KUKA KRL program: MyProgram_048().src

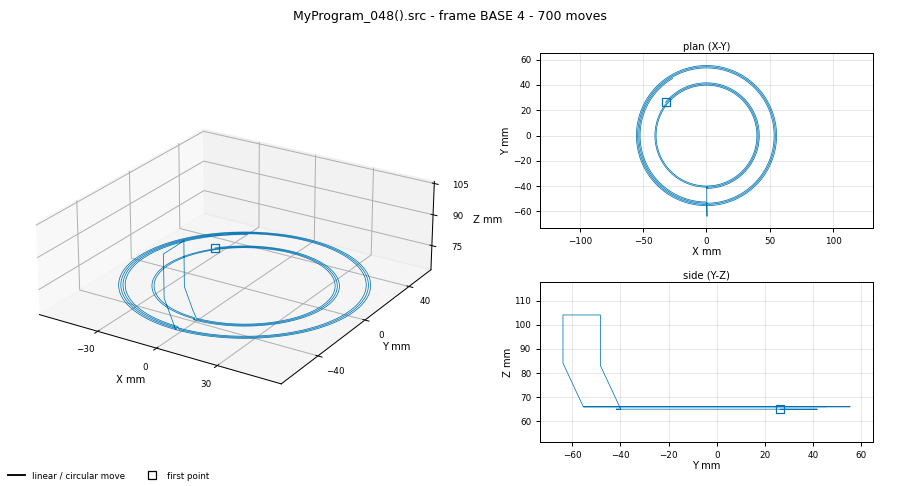
[picture p0: tool path of MyProgram_048().src in frame BASE 4, 700 of 700 moves have a stored position in this frame; points joined in program order, loops and branches not executed]
&ACCESS RVP
&REL 1
&PARAM TEMPLATE = C:\KRC\Roboter\Template\vorgabe
&PARAM EDITMASK = *
DEF MyProgram_048()
; ---- Setting reference (Base) ----
$BASE = BASE_DATA[4]

; --------------------------
; ---- Setting tool (TCP) ----
$TOOL = TOOL_DATA[3]
; --------------------------

$VEL.CP = VEL_APROX_PRINT
Startdeposition()
$VEL.CP = VEL_PRINT
LIN {X -32.3205,Y 26.3963,Z 65,A 132.8032,B 24.8389,C -2.9281,E1 24.8778,E2 -49.5424} C_DIS
LIN {X -30.8175,Y 28.1363,Z 65,A 129.9758,B 24.8376,C -2.9396,E1 24.8831,E2 -46.7299} C_DIS
LIN {X -29.3729,Y 29.641,Z 65,A 126.9235,B 24.8371,C -2.9443,E1 24.889,E2 -43.6757} C_DIS
LIN {X -27.5809,Y 31.3158,Z 65,A 123.4844,B 24.8363,C -2.951,E1 24.8961,E2 -40.2389} C_DIS
LIN {X -25.6579,Y 32.9102,Z 65,A 120.0277,B 24.8356,C -2.9579,E1 24.9037,E2 -36.7858} C_DIS
LIN {X -22.8662,Y 34.9072,Z 65,A 115.1658,B 24.8347,C -2.9653,E1 24.9148,E2 -31.9251} C_DIS
LIN {X -20.5395,Y 36.3254,Z 65,A 111.0714,B 24.8345,C -2.9676,E1 24.9247,E2 -27.824} C_DIS
LIN {X -17.2944,Y 37.9774,Z 65,A 106.8541,B 24.8325,C -2.9849,E1 24.9352,E2 -23.6369} C_DIS
LIN {X -15.0192,Y 38.9331,Z 65,A 102.7286,B 24.8331,C -2.9804,E1 24.946,E2 -19.4915} C_DIS
LIN {X -12.6961,Y 39.7516,Z 65,A 99.3773,B 24.8326,C -2.9847,E1 24.9548,E2 -16.1444} C_DIS
LIN {X -10.2597,Y 40.4489,Z 65,A 96.7038,B 24.831,C -2.9984,E1 24.962,E2 -13.4995} C_DIS
LIN {X -8.3518,Y 40.8853,Z 65,A 93.3297,B 24.8318,C -2.9918,E1 24.9712,E2 -10.1056} C_DIS
LIN {X -5.0291,Y 41.4254,Z 65,A 88.9173,B 24.8311,C -2.9975,E1 24.9834,E2 -5.7032} C_DIS
LIN {X -2.4514,Y 41.657,Z 65,A 85.2136,B 24.8311,C -2.9971,E1 24.9937,E2 -1.9969} C_DIS
LIN {X -0.4444,Y 41.7276,Z 65,A 82.0555,B 24.8317,C -2.9923,E1 25.0026,E2 1.1727} C_DIS
LIN {X 3.7427,Y 41.5615,Z 65,A 77.3936,B 24.83,C -3.0075,E1 25.0155,E2 5.7968} C_DIS
LIN {X 5.9938,Y 41.297,Z 65,A 73.4068,B 24.8315,C -2.9945,E1 25.0266,E2 9.8111} C_DIS
LIN {X 8.6502,Y 40.8239,Z 65,A 69.8403,B 24.8315,C -2.9949,E1 25.0363,E2 13.3725} C_DIS
LIN {X 11.6644,Y 40.0663,Z 65,A 65.7716,B 24.8314,C -2.9951,E1 25.0473,E2 17.4342} C_DIS
LIN {X 14.4066,Y 39.164,Z 65,A 62.3461,B 24.8309,C -2.9997,E1 25.0563,E2 20.8419} C_DIS
LIN {X 15.9978,Y 38.5419,Z 65,A 59.5196,B 24.8319,C -2.9903,E1 25.0636,E2 23.6845} C_DIS
LIN {X 19.3949,Y 36.9485,Z 65,A 55.141,B 24.8313,C -2.9959,E1 25.0746,E2 28.0383} C_DIS
LIN {X 21.1243,Y 35.988,Z 65,A 51.5538,B 24.8332,C -2.9788,E1 25.0834,E2 31.6554} C_DIS
LIN {X 23.0276,Y 34.8007,Z 65,A 48.6817,B 24.8334,C -2.9773,E1 25.0901,E2 34.5218} C_DIS
LIN {X 24.9284,Y 33.4655,Z 65,A 45.4862,B 24.834,C -2.9719,E1 25.0974,E2 37.7189} C_DIS
LIN {X 26.8036,Y 31.9836,Z 65,A 42.1697,B 24.8347,C -2.9653,E1 25.1046,E2 41.0384} C_DIS
LIN {X 28.6861,Y 30.3064,Z 65,A 38.7348,B 24.8355,C -2.9589,E1 25.1116,E2 44.4745} C_DIS
LIN {X 30.3503,Y 28.6394,Z 65,A 35.6045,B 24.836,C -2.9538,E1 25.1177,E2 47.6035} C_DIS
LIN {X 31.8657,Y 26.9436,Z 65,A 32.0272,B 24.8376,C -2.9395,E1 25.1243,E2 51.1986} C_DIS
LIN {X 33.4817,Y 24.9072,Z 65,A 28.9748,B 24.8376,C -2.9395,E1 25.1294,E2 54.2366} C_DIS
LIN {X 34.85,Y 22.9529,Z 65,A 25.5823,B 24.8387,C -2.9294,E1 25.1348,E2 57.6362} C_DIS
LIN {X 35.9583,Y 21.1746,Z 65,A 22.8285,B 24.8393,C -2.924,E1 25.1388,E2 60.3887} C_DIS
LIN {X 36.8509,Y 19.5803,Z 65,A 20.2123,B 24.8403,C -2.9156,E1 25.1423,E2 63.0112} C_DIS
LIN {X 38.143,Y 16.9264,Z 65,A 16.3814,B 24.8411,C -2.9081,E1 25.1468,E2 66.839} C_DIS
LIN {X 38.9023,Y 15.0995,Z 65,A 13.8688,B 24.8416,C -2.9039,E1 25.1494,E2 69.3479} C_DIS
LIN {X 39.6903,Y 12.8856,Z 65,A 10.013,B 24.8437,C -2.8839,E1 25.1529,E2 73.2292} C_DIS
LIN {X 40.4156,Y 10.3892,Z 65,A 7.2043,B 24.8435,C -2.8862,E1 25.155,E2 76.0163} C_DIS
LIN {X 40.9346,Y 8.1069,Z 65,A 3.7683,B 24.845,C -2.8727,E1 25.1571,E2 79.4643} C_DIS
LIN {X 41.2614,Y 6.2336,Z 65,A 1.2108,B 24.8457,C -2.8656,E1 25.1582,E2 82.0235} C_DIS
LIN {X 41.531,Y 4.0697,Z 65,A -2.1598,B 24.8474,C -2.8499,E1 25.1593,E2 85.4114} C_DIS
LIN {X 41.6995,Y 1.5955,Z 65,A -5.1201,B 24.8477,C -2.8469,E1 25.1597,E2 88.3612} C_DIS
LIN {X 41.7291,Y 0.1295,Z 65,A -7.4448,B 24.849,C -2.8352,E1 25.1597,E2 90.6997} C_DIS
LIN {X 41.6403,Y -2.7296,Z 65,A -11.1427,B 24.8499,C -2.8268,E1 25.1593,E2 94.3955} C_DIS
LIN {X 41.4605,Y -4.7326,Z 65,A -13.8628,B 24.8507,C -2.8188,E1 25.1585,E2 97.1184} C_DIS
LIN {X 41.1292,Y -7.0549,Z 65,A -17.206,B 24.852,C -2.8066,E1 25.1571,E2 100.4708} C_DIS
LIN {X 40.6295,Y -9.5191,Z 65,A -20.7553,B 24.8533,C -2.7942,E1 25.155,E2 104.0287} C_DIS
LIN {X 39.9708,Y -11.9877,Z 65,A -24.0951,B 24.8542,C -2.7863,E1 25.1524,E2 107.3682} C_DIS
LIN {X 39.1708,Y -14.3878,Z 65,A -27.523,B 24.8552,C -2.7766,E1 25.1493,E2 110.7999} C_DIS
LIN {X 38.33,Y -16.4987,Z 65,A -30.7347,B 24.8563,C -2.7657,E1 25.1458,E2 114.0196} C_DIS
LIN {X 37.2921,Y -18.727,Z 65,A -34.2725,B 24.8576,C -2.7531,E1 25.1415,E2 117.5684} C_DIS
LIN {X 35.9701,Y -21.1546,Z 65,A -37.5233,B 24.8578,C -2.7515,E1 25.1371,E2 120.806} C_DIS
LIN {X 35.1122,Y -22.5497,Z 65,A -40.3199,B 24.8594,C -2.736,E1 25.1329,E2 123.625} C_DIS
LIN {X 33.0565,Y -25.4681,Z 65,A -44.5679,B 24.8596,C -2.7339,E1 25.1259,E2 127.8576} C_DIS
LIN {X 30.9077,Y -28.0379,Z 65,A -50.2918,B 24.8627,C -2.7037,E1 25.1154,E2 133.6271} C_DIS
LIN {X 27.7752,Y -31.1432,Z 65,A -56.1001,B 24.8637,C -2.6938,E1 25.1036,E2 139.4351} C_DIS
LIN {X 25.3244,Y -33.1672,Z 65,A -60.489,B 24.8647,C -2.6842,E1 25.0939,E2 143.8306} C_DIS
LIN {X 22.261,Y -35.2964,Z 65,A -64.6735,B 24.8642,C -2.6892,E1 25.0842,E2 147.9891} C_DIS
LIN {X 20.7403,Y -36.2105,Z 65,A -67.3879,B 24.8651,C -2.6804,E1 25.0777,E2 150.7159} C_DIS
LIN {X 18.6693,Y -37.3207,Z 65,A -70.5143,B 24.8655,C -2.6767,E1 25.0699,E2 153.8425} C_DIS
LIN {X 16.6026,Y -38.2847,Z 65,A -73.9067,B 24.8663,C -2.668,E1 25.0613,E2 157.2473} C_DIS
LIN {X 14.2014,Y -39.2388,Z 65,A -77.1234,B 24.8663,C -2.6683,E1 25.0529,E2 160.4561} C_DIS
LIN {X 12.1209,Y -39.9312,Z 65,A -80.2732,B 24.8669,C -2.6627,E1 25.0445,E2 163.6136} C_DIS
LIN {X 9.9555,Y -40.5247,Z 65,A -83.3276,B 24.8671,C -2.66,E1 25.0362,E2 166.6696} C_DIS
LIN {X 7.6108,Y -41.0292,Z 65,A -86.1957,B 24.8668,C -2.6636,E1 25.0284,E2 169.5257} C_DIS
LIN {X 6.2927,Y -41.2524,Z 65,A -88.5034,B 24.8676,C -2.6553,E1 25.022,E2 171.8509} C_DIS
LIN {X 4.1311,Y -41.525,Z 65,A -91.2129,B 24.8674,C -2.6577,E1 25.0145,E2 174.5529} C_DIS
LIN {X 2.1588,Y -41.6739,Z 65,A -94.0601,B 24.8677,C -2.6546,E1 25.0065,E2 177.4061} C_DIS
LIN {X 0.2084,Y -41.7255,Z 65,A -95.7171,B 24.8663,C -2.6686,E1 25.002,E2 179.0294} C_DIS
Enddeposition()
LIN {X 0.2084,Y -41.7255,Z 65,A -95.7171,B 24.8663,C -2.6686,E1 25.002,E2 179.0294} C_DIS
Startdeposition()
$VEL.CP = VEL_PRINT
LIN {X 0.7849,Y -40.7795,Z 65,A -94.3839,B 24.8639,C -2.6925,E1 25.0059,E2 177.6397} C_DIS
LIN {X 3.4989,Y -40.6375,Z 65,A -90.8703,B 24.8641,C -2.6897,E1 25.0157,E2 174.1342} C_DIS
LIN {X 5.4478,Y -40.4216,Z 65,A -88.0105,B 24.8638,C -2.6929,E1 25.0236,E2 171.2689} C_DIS
LIN {X 7.6059,Y -40.0718,Z 65,A -84.7696,B 24.8633,C -2.6978,E1 25.0325,E2 168.0199} C_DIS
LIN {X 10.1651,Y -39.5001,Z 65,A -81.273,B 24.8633,C -2.6985,E1 25.042,E2 164.5267} C_DIS
LIN {X 12.8249,Y -38.7189,Z 65,A -76.8382,B 24.8619,C -2.7113,E1 25.0539,E2 160.0697} C_DIS
LIN {X 15.5731,Y -37.6976,Z 65,A -73.1485,B 24.8621,C -2.7102,E1 25.0635,E2 156.3906} C_DIS
LIN {X 17.805,Y -36.6959,Z 65,A -69.8338,B 24.8617,C -2.7136,E1 25.0718,E2 153.0764} C_DIS
LIN {X 19.7266,Y -35.6999,Z 65,A -66.6692,B 24.861,C -2.7206,E1 25.0797,E2 149.9041} C_DIS
LIN {X 21.6021,Y -34.5967,Z 65,A -63.8109,B 24.8607,C -2.7231,E1 25.0865,E2 147.049} C_DIS
LIN {X 23.9097,Y -33.0449,Z 65,A -59.7045,B 24.8596,C -2.734,E1 25.0959,E2 142.9308} C_DIS
LIN {X 25.861,Y -31.5412,Z 65,A -56.2483,B 24.8589,C -2.7413,E1 25.1035,E2 139.4702} C_DIS
LIN {X 27.7138,Y -29.926,Z 65,A -53.35,B 24.8589,C -2.74,E1 25.1095,E2 136.5865} C_DIS
LIN {X 28.9865,Y -28.6944,Z 65,A -50.4742,B 24.8577,C -2.7523,E1 25.1152,E2 133.6937} C_DIS
LIN {X 30.4702,Y -27.1136,Z 65,A -47.0406,B 24.8563,C -2.7663,E1 25.1217,E2 130.2422} C_DIS
LIN {X 32.3443,Y -24.8482,Z 65,A -43.3381,B 24.8559,C -2.7698,E1 25.1281,E2 126.5486} C_DIS
LIN {X 33.6292,Y -23.0807,Z 65,A -40.4032,B 24.8553,C -2.7758,E1 25.1329,E2 123.6139} C_DIS
LIN {X 34.9472,Y -21.0305,Z 65,A -36.6735,B 24.8537,C -2.7905,E1 25.1384,E2 119.8682} C_DIS
LIN {X 35.9255,Y -19.3122,Z 65,A -34.0007,B 24.8531,C -2.7966,E1 25.142,E2 117.1948} C_DIS
LIN {X 37.0399,Y -17.0779,Z 65,A -30.6076,B 24.8522,C -2.805,E1 25.1461,E2 113.8003} C_DIS
LIN {X 37.907,Y -15.0554,Z 65,A -27.4857,B 24.8512,C -2.8147,E1 25.1494,E2 110.6725} C_DIS
LIN {X 38.6802,Y -12.9398,Z 65,A -24.7937,B 24.851,C -2.8162,E1 25.1519,E2 107.992} C_DIS
LIN {X 39.2211,Y -11.1934,Z 65,A -22.2257,B 24.8502,C -2.8241,E1 25.154,E2 105.42} C_DIS
LIN {X 39.6949,Y -9.3771,Z 65,A -19.2563,B 24.8487,C -2.838,E1 25.156,E2 102.435} C_DIS
LIN {X 40.1515,Y -7.1725,Z 65,A -16.0267,B 24.8475,C -2.849,E1 25.1577,E2 99.1981} C_DIS
LIN {X 40.5125,Y -4.7251,Z 65,A -12.5987,B 24.8464,C -2.8591,E1 25.159,E2 95.7665} C_DIS
LIN {X 40.7053,Y -2.5869,Z 65,A -9.1965,B 24.8447,C -2.8752,E1 25.1596,E2 92.3463} C_DIS
LIN {X 40.776,Y 0.949,Z 65,A -4.9181,B 24.8443,C -2.8789,E1 25.1596,E2 88.0845} C_DIS
LIN {X 40.615,Y 3.7424,Z 65,A -0.3025,B 24.8417,C -2.9029,E1 25.1587,E2 83.4396} C_DIS
LIN {X 40.2879,Y 6.363,Z 65,A 3.1785,B 24.8408,C -2.9104,E1 25.1573,E2 79.9614} C_DIS
LIN {X 39.6611,Y 9.5174,Z 65,A 7.3091,B 24.8401,C -2.9174,E1 25.1549,E2 75.8382} C_DIS
LIN {X 39.038,Y 11.8165,Z 65,A 10.7303,B 24.8388,C -2.9286,E1 25.1523,E2 72.4102} C_DIS
LIN {X 38.4737,Y 13.5412,Z 65,A 12.883,B 24.8388,C -2.9293,E1 25.1503,E2 70.2679} C_DIS
LIN {X 37.9097,Y 15.0486,Z 65,A 15.4724,B 24.8374,C -2.9413,E1 25.1477,E2 67.6645} C_DIS
LIN {X 36.8271,Y 17.532,Z 65,A 19.3626,B 24.8361,C -2.9532,E1 25.1432,E2 63.7671} C_DIS
LIN {X 35.7144,Y 19.7005,Z 65,A 22.6885,B 24.8353,C -2.9607,E1 25.1388,E2 60.441} C_DIS
LIN {X 34.6226,Y 21.5607,Z 65,A 25.3115,B 24.8351,C -2.9618,E1 25.1351,E2 57.8287} C_DIS
LIN {X 33.0626,Y 23.8852,Z 65,A 29.4017,B 24.8338,C -2.9741,E1 25.1286,E2 53.7296} C_DIS
LIN {X 32.106,Y 25.1559,Z 65,A 32.0073,B 24.8325,C -2.9854,E1 25.1241,E2 51.1095} C_DIS
LIN {X 30.2152,Y 27.3986,Z 65,A 36.0076,B 24.8317,C -2.9927,E1 25.1168,E2 47.1101} C_DIS
LIN {X 28.5261,Y 29.1528,Z 65,A 39.37,B 24.831,C -2.9989,E1 25.1102,E2 43.7473} C_DIS
LIN {X 26.7641,Y 30.7779,Z 65,A 42.6418,B 24.8304,C -3.0039,E1 25.1034,E2 40.4767} C_DIS
LIN {X 24.9657,Y 32.2538,Z 65,A 45.9762,B 24.8296,C -3.0108,E1 25.0961,E2 37.1383} C_DIS
LIN {X 22.9381,Y 33.7259,Z 65,A 49.302,B 24.8293,C -3.0136,E1 25.0885,E2 33.8175} C_DIS
LIN {X 21.1922,Y 34.8494,Z 65,A 52.6119,B 24.8281,C -3.024,E1 25.0806,E2 30.4934} C_DIS
LIN {X 18.538,Y 36.3308,Z 65,A 56.2779,B 24.8285,C -3.0204,E1 25.0717,E2 26.8464} C_DIS
LIN {X 16.757,Y 37.1859,Z 65,A 59.369,B 24.8276,C -3.0283,E1 25.0638,E2 23.7444} C_DIS
LIN {X 14.6433,Y 38.0684,Z 65,A 62.6886,B 24.8271,C -3.033,E1 25.0552,E2 20.4212} C_DIS
LIN {X 12.286,Y 38.8933,Z 65,A 65.5956,B 24.8278,C -3.027,E1 25.0475,E2 17.5339} C_DIS
LIN {X 10.6833,Y 39.3631,Z 65,A 69.197,B 24.8255,C -3.0468,E1 25.0377,E2 13.8914} C_DIS
LIN {X 7.2645,Y 40.135,Z 65,A 73.3488,B 24.8265,C -3.0378,E1 25.0265,E2 9.7661} C_DIS
LIN {X 4.9873,Y 40.4811,Z 65,A 76.4292,B 24.8267,C -3.0364,E1 25.0179,E2 6.6917} C_DIS
LIN {X 3.2904,Y 40.6541,Z 65,A 78.7021,B 24.8269,C -3.0349,E1 25.0116,E2 4.4237} C_DIS
LIN {X 1.2643,Y 40.7675,Z 65,A 82.277,B 24.8257,C -3.0447,E1 25.0016,E2 0.8265} C_DIS
LIN {X -1.7811,Y 40.7482,Z 65,A 86.121,B 24.8266,C -3.0376,E1 24.9909,E2 -3.0011} C_DIS
LIN {X -4.2792,Y 40.562,Z 65,A 90.6441,B 24.8252,C -3.0494,E1 24.9783,E2 -7.5547} C_DIS
LIN {X -8.1041,Y 39.974,Z 65,A 95.7175,B 24.8262,C -3.0404,E1 24.9644,E2 -12.6121} C_DIS
LIN {X -11.7877,Y 39.0471,Z 65,A 100.4469,B 24.8277,C -3.0272,E1 24.9517,E2 -17.3172} C_DIS
LIN {X -14.0402,Y 38.2944,Z 65,A 103.7453,B 24.8283,C -3.0227,E1 24.943,E2 -20.6112} C_DIS
LIN {X -15.9024,Y 37.5593,Z 65,A 106.1998,B 24.8292,C -3.0144,E1 24.9367,E2 -23.0515} C_DIS
LIN {X -18.3667,Y 36.4184,Z 65,A 111.1925,B 24.8282,C -3.023,E1 24.9241,E2 -28.0776} C_DIS
LIN {X -21.3412,Y 34.7588,Z 65,A 115.2173,B 24.8302,C -3.0054,E1 24.9145,E2 -32.0725} C_DIS
LIN {X -23.457,Y 33.3676,Z 65,A 118.8869,B 24.8309,C -2.9999,E1 24.906,E2 -35.7413} C_DIS
LIN {X -25.4735,Y 31.855,Z 65,A 122.4407,B 24.8317,C -2.9927,E1 24.8982,E2 -39.2909} C_DIS
LIN {X -27.3021,Y 30.3017,Z 65,A 125.7452,B 24.8326,C -2.9845,E1 24.8912,E2 -42.5888} C_DIS
LIN {X -29.076,Y 28.6039,Z 65,A 128.9546,B 24.8338,C -2.9737,E1 24.8849,E2 -45.7859} C_DIS
LIN {X -30.3502,Y 27.248,Z 65,A 131.9306,B 24.8341,C -2.9715,E1 24.8792,E2 -48.7696} C_DIS
LIN {X -31.9657,Y 25.3334,Z 65,A 135.4098,B 24.8351,C -2.962,E1 24.8731,E2 -52.2424} C_DIS
LIN {X -33.3945,Y 23.4184,Z 65,A 138.8033,B 24.8361,C -2.9535,E1 24.8676,E2 -55.6321} C_DIS
LIN {X -34.7081,Y 21.4239,Z 65,A 142.1037,B 24.8372,C -2.9437,E1 24.8626,E2 -58.9257} C_DIS
LIN {X -35.7924,Y 19.5577,Z 65,A 145.1702,B 24.8381,C -2.9355,E1 24.8584,E2 -61.9887} C_DIS
LIN {X -36.8745,Y 17.4332,Z 65,A 148.3179,B 24.8394,C -2.9236,E1 24.8545,E2 -65.1249} C_DIS
LIN {X -37.9062,Y 15.0576,Z 65,A 152.2189,B 24.8403,C -2.9157,E1 24.8503,E2 -69.0285} C_DIS
LIN {X -38.711,Y 12.8484,Z 65,A 155.4631,B 24.8414,C -2.9051,E1 24.8473,E2 -72.2657} C_DIS
LIN {X -39.3303,Y 10.8047,Z 65,A 158.6925,B 24.8422,C -2.8984,E1 24.8448,E2 -75.4977} C_DIS
LIN {X -39.881,Y 8.5504,Z 65,A 161.5006,B 24.8438,C -2.8834,E1 24.8431,E2 -78.2865} C_DIS
LIN {X -40.1774,Y 7.0287,Z 65,A 164.2148,B 24.8438,C -2.8824,E1 24.8417,E2 -81.0143} C_DIS
LIN {X -40.5153,Y 4.7009,Z 65,A 167.0069,B 24.8456,C -2.8666,E1 24.8407,E2 -83.7852} C_DIS
LIN {X -40.7269,Y 2.2152,Z 65,A 170.9567,B 24.8463,C -2.8603,E1 24.8399,E2 -87.7438} C_DIS
LIN {X -40.7865,Y -0.2829,Z 65,A 174.5588,B 24.8474,C -2.8503,E1 24.8399,E2 -91.3436} C_DIS
LIN {X -40.6844,Y -2.8956,Z 65,A 178.0933,B 24.8488,C -2.8374,E1 24.8404,E2 -94.8684} C_DIS
LIN {X -40.5292,Y -4.5821,Z 65,A -179.3218,B 24.8493,C -2.8322,E1 24.8411,E2 -97.4565} C_DIS
LIN {X -40.0876,Y -7.5239,Z 65,A -175.1297,B 24.8507,C -2.8196,E1 24.8431,E2 -101.6433} C_DIS
LIN {X -39.5764,Y -9.8657,Z 65,A -171.9067,B 24.8519,C -2.8079,E1 24.8451,E2 -104.8573} C_DIS
LIN {X -38.9417,Y -12.1297,Z 65,A -168.9289,B 24.8533,C -2.7946,E1 24.8474,E2 -107.8205} C_DIS
LIN {X -38.2219,Y -14.2365,Z 65,A -165.2743,B 24.8536,C -2.7914,E1 24.8508,E2 -111.4882} C_DIS
LIN {X -37.2883,Y -16.5297,Z 65,A -161.827,B 24.8547,C -2.7813,E1 24.8546,E2 -114.9305} C_DIS
LIN {X -36.2762,Y -18.6448,Z 65,A -158.6127,B 24.8557,C -2.7715,E1 24.8586,E2 -118.1386} C_DIS
LIN {X -34.9175,Y -21.0801,Z 65,A -154.5325,B 24.8566,C -2.7632,E1 24.8643,E2 -122.22} C_DIS
LIN {X -33.6067,Y -23.1131,Z 65,A -151.0904,B 24.8574,C -2.7552,E1 24.8696,E2 -125.6603} C_DIS
LIN {X -32.3412,Y -24.8523,Z 65,A -147.9387,B 24.858,C -2.7496,E1 24.8749,E2 -128.8136} C_DIS
LIN {X -30.5769,Y -26.9934,Z 65,A -144.1509,B 24.859,C -2.7395,E1 24.8818,E2 -132.5947} C_DIS
LIN {X -28.8359,Y -28.8467,Z 65,A -140.555,B 24.8598,C -2.7323,E1 24.8888,E2 -136.1889} C_DIS
LIN {X -27.004,Y -30.5683,Z 65,A -137.4763,B 24.8611,C -2.72,E1 24.8951,E2 -139.2506} C_DIS
LIN {X -25.0502,Y -32.1887,Z 65,A -133.4236,B 24.8611,C -2.7195,E1 24.9039,E2 -143.3172} C_DIS
LIN {X -23.4292,Y -33.387,Z 65,A -130.3144,B 24.8612,C -2.7183,E1 24.911,E2 -146.4345} C_DIS
LIN {X -20.8855,Y -35.0342,Z 65,A -126.1779,B 24.862,C -2.7106,E1 24.9208,E2 -150.5654} C_DIS
LIN {X -18.5001,Y -36.3502,Z 65,A -122.6394,B 24.8629,C -2.702,E1 24.9295,E2 -154.0934} C_DIS
LIN {X -16.6041,Y -37.2548,Z 65,A -119.5679,B 24.8631,C -2.7003,E1 24.9373,E2 -157.1684} C_DIS
LIN {X -14.3986,Y -38.1611,Z 65,A -116.44,B 24.8637,C -2.6943,E1 24.9454,E2 -160.2887} C_DIS
LIN {X -11.2696,Y -39.1996,Z 65,A -111.5093,B 24.8637,C -2.6948,E1 24.9585,E2 -165.2295} C_DIS
LIN {X -8.4128,Y -39.9106,Z 65,A -107.1405,B 24.8635,C -2.696,E1 24.9704,E2 -169.6068} C_DIS
LIN {X -4.7607,Y -40.5083,Z 65,A -101.7408,B 24.8633,C -2.6977,E1 24.9854,E2 -175.0148} C_DIS
LIN {X -2.1707,Y -40.7293,Z 65,A -98.2739,B 24.8636,C -2.6952,E1 24.995,E2 -178.477} C_DIS
LIN {X 0.2059,Y -40.781,Z 65,A -96.1977,B 24.8653,C -2.678,E1 25.0007,E2 -180.5123} C_DIS
Enddeposition()
LIN {X 0.2059,Y -40.781,Z 65,A -96.1977,B 24.8653,C -2.678,E1 25.0007,E2 -180.5123} C_DIS
Startdeposition()
$VEL.CP = VEL_PRINT
LIN {X -0.4047,Y -39.8429,Z 65,A -97.6468,B 24.8645,C -2.6863,E1 24.9967,E2 -179.0829} C_DIS
LIN {X -2.4418,Y -39.7704,Z 65,A -100.789,B 24.8648,C -2.6832,E1 24.988,E2 -175.9327} C_DIS
LIN {X -4.8574,Y -39.548,Z 65,A -104.0622,B 24.8645,C -2.6864,E1 24.9789,E2 -172.6651} C_DIS
LIN {X -6.9556,Y -39.2329,Z 65,A -107.3,B 24.8646,C -2.6849,E1 24.9699,E2 -169.4206} C_DIS
LIN {X -9.2215,Y -38.7635,Z 65,A -110.5774,B 24.8644,C -2.687,E1 24.961,E2 -166.1442} C_DIS
LIN {X -11.4617,Y -38.1607,Z 65,A -113.8715,B 24.8641,C -2.6897,E1 24.9522,E2 -162.8512} C_DIS
LIN {X -13.441,Y -37.5097,Z 65,A -116.8946,B 24.8639,C -2.6918,E1 24.9442,E2 -159.8272} C_DIS
LIN {X -15.612,Y -36.659,Z 65,A -120.1596,B 24.8635,C -2.6961,E1 24.9357,E2 -156.5653} C_DIS
LIN {X -17.4806,Y -35.8061,Z 65,A -123.1197,B 24.8632,C -2.6994,E1 24.9283,E2 -153.6054} C_DIS
LIN {X -19.3027,Y -34.8571,Z 65,A -126.3038,B 24.8631,C -2.7004,E1 24.9204,E2 -150.4149} C_DIS
LIN {X -21.3397,Y -33.649,Z 65,A -129.5918,B 24.8624,C -2.7067,E1 24.9126,E2 -147.1317} C_DIS
LIN {X -23.2623,Y -32.3493,Z 65,A -132.8971,B 24.8618,C -2.7125,E1 24.905,E2 -143.8289} C_DIS
LIN {X -25.0817,Y -30.9596,Z 65,A -136.3096,B 24.8614,C -2.7169,E1 24.8975,E2 -140.4143} C_DIS
LIN {X -26.9039,Y -29.39,Z 65,A -139.7827,B 24.8607,C -2.7233,E1 24.8903,E2 -136.9429} C_DIS
LIN {X -28.5561,Y -27.788,Z 65,A -143.142,B 24.8601,C -2.7296,E1 24.8837,E2 -133.5843} C_DIS
LIN {X -29.7107,Y -26.5493,Z 65,A -145.5464,B 24.8595,C -2.7352,E1 24.8792,E2 -131.1827} C_DIS
LIN {X -31.2399,Y -24.7318,Z 65,A -148.9577,B 24.8587,C -2.7431,E1 24.8731,E2 -127.7743} C_DIS
LIN {X -32.5816,Y -22.9366,Z 65,A -152.1759,B 24.8579,C -2.7509,E1 24.8679,E2 -124.5591} C_DIS
LIN {X -33.865,Y -20.9945,Z 65,A -155.4949,B 24.857,C -2.7596,E1 24.8629,E2 -121.2443} C_DIS
LIN {X -34.9596,Y -19.1164,Z 65,A -158.7885,B 24.8563,C -2.766,E1 24.8583,E2 -117.9487} C_DIS
LIN {X -35.9694,Y -17.1409,Z 65,A -161.8615,B 24.8553,C -2.7759,E1 24.8545,E2 -114.8828} C_DIS
LIN {X -36.851,Y -15.1531,Z 65,A -165.1616,B 24.8545,C -2.7829,E1 24.8509,E2 -111.5811} C_DIS
LIN {X -37.649,Y -13.0447,Z 65,A -168.2143,B 24.8533,C -2.7941,E1 24.848,E2 -108.538} C_DIS
LIN {X -38.2712,Y -11.0889,Z 65,A -171.1844,B 24.8525,C -2.8026,E1 24.8456,E2 -105.571} C_DIS
LIN {X -38.7677,Y -9.2043,Z 65,A -174.1068,B 24.8517,C -2.8097,E1 24.8436,E2 -102.6487} C_DIS
LIN {X -39.2391,Y -6.9209,Z 65,A -177.399,B 24.8506,C -2.8205,E1 24.8419,E2 -99.3628} C_DIS
LIN {X -39.5597,Y -4.7582,Z 65,A 179.2576,B 24.8497,C -2.8282,E1 24.8407,E2 -96.0178} C_DIS
LIN {X -39.7707,Y -2.4366,Z 65,A 176.0727,B 24.8484,C -2.8403,E1 24.84,E2 -92.8427} C_DIS
LIN {X -39.8441,Y -0.2609,Z 65,A 172.753,B 24.8476,C -2.8482,E1 24.8398,E2 -89.5218} C_DIS
LIN {X -39.792,Y 2.0526,Z 65,A 169.4211,B 24.8465,C -2.8586,E1 24.8401,E2 -86.1948} C_DIS
LIN {X -39.6132,Y 4.2905,Z 65,A 166.2657,B 24.8453,C -2.8694,E1 24.8409,E2 -83.0465} C_DIS
LIN {X -39.3195,Y 6.4484,Z 65,A 162.9682,B 24.8444,C -2.8776,E1 24.8423,E2 -79.7488} C_DIS
LIN {X -38.8981,Y 8.6341,Z 65,A 159.9339,B 24.8432,C -2.8892,E1 24.844,E2 -76.7243} C_DIS
LIN {X -38.4293,Y 10.5261,Z 65,A 157.1107,B 24.8422,C -2.8976,E1 24.846,E2 -73.9049} C_DIS
LIN {X -37.8363,Y 12.4926,Z 65,A 154.1355,B 24.8413,C -2.9064,E1 24.8485,E2 -70.9336} C_DIS
LIN {X -37.1422,Y 14.4248,Z 65,A 150.9639,B 24.8405,C -2.913,E1 24.8516,E2 -67.76} C_DIS
LIN {X -36.1926,Y 16.6648,Z 65,A 147.4209,B 24.8395,C -2.9229,E1 24.8556,E2 -64.2211} C_DIS
LIN {X -35.1423,Y 18.7794,Z 65,A 144.108,B 24.8383,C -2.9335,E1 24.8598,E2 -60.9159} C_DIS
LIN {X -33.9723,Y 20.8205,Z 65,A 140.8154,B 24.8371,C -2.9439,E1 24.8645,E2 -57.6311} C_DIS
LIN {X -32.8535,Y 22.5454,Z 65,A 137.8412,B 24.8363,C -2.9517,E1 24.8691,E2 -54.6608} C_DIS
LIN {X -31.5614,Y 24.3201,Z 65,A 134.5264,B 24.8355,C -2.9583,E1 24.8746,E2 -51.3459} C_DIS
LIN {X -30.014,Y 26.2059,Z 65,A 130.9805,B 24.8346,C -2.9668,E1 24.881,E2 -47.8039} C_DIS
LIN {X -28.3408,Y 28.007,Z 65,A 127.4412,B 24.8336,C -2.9752,E1 24.8878,E2 -44.2695} C_DIS
LIN {X -26.5741,Y 29.6885,Z 65,A 123.9167,B 24.8328,C -2.983,E1 24.8951,E2 -40.7493} C_DIS
LIN {X -24.7489,Y 31.2264,Z 65,A 120.4789,B 24.8319,C -2.9902,E1 24.9025,E2 -37.3158} C_DIS
LIN {X -22.9495,Y 32.5725,Z 65,A 117.2622,B 24.8312,C -2.9968,E1 24.9097,E2 -34.1037} C_DIS
LIN {X -20.9872,Y 33.8696,Z 65,A 113.9099,B 24.8305,C -3.0035,E1 24.9176,E2 -30.7564} C_DIS
LIN {X -19.0694,Y 34.9851,Z 65,A 110.5857,B 24.83,C -3.0074,E1 24.9257,E2 -27.4318} C_DIS
LIN {X -17.1026,Y 35.9878,Z 65,A 107.5121,B 24.8293,C -3.0135,E1 24.9334,E2 -24.3647} C_DIS
LIN {X -15.1345,Y 36.8585,Z 65,A 104.2773,B 24.829,C -3.0162,E1 24.9417,E2 -21.1289} C_DIS
LIN {X -12.8582,Y 37.7131,Z 65,A 100.7661,B 24.8285,C -3.0203,E1 24.9509,E2 -17.6206} C_DIS
LIN {X -10.7348,Y 38.3715,Z 65,A 97.7351,B 24.8279,C -3.0258,E1 24.959,E2 -14.5976} C_DIS
LIN {X -8.8159,Y 38.8574,Z 65,A 94.7529,B 24.8279,C -3.0267,E1 24.9671,E2 -11.6136} C_DIS
LIN {X -6.3949,Y 39.3285,Z 65,A 91.287,B 24.8274,C -3.0303,E1 24.9766,E2 -8.1528} C_DIS
LIN {X -4.3696,Y 39.6049,Z 65,A 88.3107,B 24.8272,C -3.0316,E1 24.9849,E2 -5.1774} C_DIS
LIN {X -2.0522,Y 39.792,Z 65,A 85.0093,B 24.827,C -3.0335,E1 24.9941,E2 -1.8792} C_DIS
LIN {X -0.0033,Y 39.8453,Z 65,A 82.0298,B 24.827,C -3.0337,E1 25.0024,E2 1.0998} C_DIS
LIN {X 2.1171,Y 39.7884,Z 65,A 78.8858,B 24.8271,C -3.0327,E1 25.0111,E2 4.2453} C_DIS
LIN {X 4.3168,Y 39.6104,Z 65,A 75.8295,B 24.827,C -3.0339,E1 25.0196,E2 7.2968} C_DIS
LIN {X 6.4445,Y 39.3202,Z 65,A 72.6088,B 24.8273,C -3.0313,E1 25.0285,E2 10.5208} C_DIS
LIN {X 8.6233,Y 38.9005,Z 65,A 69.5912,B 24.8272,C -3.0322,E1 25.0368,E2 13.5324} C_DIS
LIN {X 10.5474,Y 38.4236,Z 65,A 66.6103,B 24.8276,C -3.0287,E1 25.0448,E2 16.5171} C_DIS
LIN {X 12.8743,Y 37.7076,Z 65,A 63.1185,B 24.8279,C -3.0261,E1 25.0541,E2 20.0085} C_DIS
LIN {X 15.154,Y 36.8506,Z 65,A 59.7248,B 24.8281,C -3.0243,E1 25.0629,E2 23.399} C_DIS
LIN {X 17.0329,Y 36.0212,Z 65,A 56.701,B 24.8286,C -3.0199,E1 25.0706,E2 26.4256} C_DIS
LIN {X 19.1839,Y 34.923,Z 65,A 53.3097,B 24.829,C -3.0166,E1 25.079,E2 29.8151} C_DIS
LIN {X 21.0057,Y 33.8581,Z 65,A 50.1601,B 24.8296,C -3.0106,E1 25.0865,E2 32.9693} C_DIS
LIN {X 22.8679,Y 32.6293,Z 65,A 47.0995,B 24.83,C -3.0076,E1 25.0936,E2 36.0265} C_DIS
LIN {X 24.5209,Y 31.4065,Z 65,A 43.9952,B 24.8308,C -3.0003,E1 25.1005,E2 39.137} C_DIS
LIN {X 26.3965,Y 29.8475,Z 65,A 40.5,B 24.8315,C -2.9938,E1 25.1079,E2 42.6339} C_DIS
LIN {X 28.1734,Y 28.1764,Z 65,A 37.0087,B 24.8323,C -2.9869,E1 25.1149,E2 46.127} C_DIS
LIN {X 29.8862,Y 26.3523,Z 65,A 33.6888,B 24.8327,C -2.9834,E1 25.1211,E2 49.4406} C_DIS
LIN {X 31.2658,Y 24.699,Z 65,A 30.465,B 24.8337,C -2.9743,E1 25.1268,E2 52.6711} C_DIS
LIN {X 32.5923,Y 22.9212,Z 65,A 27.2857,B 24.8346,C -2.9667,E1 25.132,E2 55.8529} C_DIS
LIN {X 33.875,Y 20.9786,Z 65,A 23.9989,B 24.8354,C -2.9592,E1 25.137,E2 59.1409} C_DIS
LIN {X 34.96,Y 19.1156,Z 65,A 20.7778,B 24.8366,C -2.9491,E1 25.1414,E2 62.3691} C_DIS
LIN {X 35.9313,Y 17.2202,Z 65,A 17.8189,B 24.8373,C -2.9425,E1 25.1451,E2 65.3281} C_DIS
LIN {X 36.9065,Y 15.0167,Z 65,A 14.3184,B 24.8384,C -2.9322,E1 25.1489,E2 68.8337} C_DIS
LIN {X 37.7337,Y 12.7969,Z 65,A 10.9401,B 24.8395,C -2.9228,E1 25.1521,E2 72.2153} C_DIS
LIN {X 38.377,Y 10.7155,Z 65,A 7.992,B 24.8402,C -2.9166,E1 25.1544,E2 75.1612} C_DIS
LIN {X 38.8478,Y 8.8571,Z 65,A 5.2058,B 24.8411,C -2.9078,E1 25.1562,E2 77.9521} C_DIS
LIN {X 39.334,Y 6.3616,Z 65,A 1.485,B 24.8425,C -2.8956,E1 25.1581,E2 81.68} C_DIS
LIN {X 39.6105,Y 4.3158,Z 65,A -1.3965,B 24.8433,C -2.8879,E1 25.1591,E2 84.5628} C_DIS
LIN {X 39.7924,Y 2.0452,Z 65,A -4.623,B 24.8443,C -2.8785,E1 25.1597,E2 87.7924} C_DIS
LIN {X 39.8442,Y -0.2385,Z 65,A -7.9153,B 24.8455,C -2.8681,E1 25.1597,E2 91.0897} C_DIS
LIN {X 39.7782,Y -2.3007,Z 65,A -10.8621,B 24.8464,C -2.8591,E1 25.1594,E2 94.0403} C_DIS
LIN {X 39.5842,Y -4.549,Z 65,A -14.1625,B 24.8476,C -2.848,E1 25.1585,E2 97.3474} C_DIS
LIN {X 39.2415,Y -6.9077,Z 65,A -17.648,B 24.8489,C -2.8363,E1 25.1569,E2 100.8401} C_DIS
LIN {X 38.7406,Y -9.3152,Z 65,A -21.0432,B 24.8498,C -2.8276,E1 25.1548,E2 104.2361} C_DIS
LIN {X 38.1548,Y -11.4817,Z 65,A -24.187,B 24.8507,C -2.819,E1 25.1524,E2 107.3822} C_DIS
LIN {X 37.5124,Y -13.4337,Z 65,A -27.1651,B 24.8517,C -2.8097,E1 25.1497,E2 110.3657} C_DIS
LIN {X 36.6614,Y -15.6061,Z 65,A -30.4018,B 24.8526,C -2.8016,E1 25.1463,E2 113.6036} C_DIS
LIN {X 35.8082,Y -17.4764,Z 65,A -33.3386,B 24.8534,C -2.7932,E1 25.1428,E2 116.5444} C_DIS
LIN {X 34.835,Y -19.3423,Z 65,A -36.5193,B 24.8546,C -2.782,E1 25.1386,E2 119.7348} C_DIS
LIN {X 33.6507,Y -21.3371,Z 65,A -39.751,B 24.8554,C -2.7744,E1 25.1339,E2 122.9682} C_DIS
LIN {X 32.348,Y -23.2641,Z 65,A -43.0321,B 24.8563,C -2.7664,E1 25.1286,E2 126.2521} C_DIS
LIN {X 31.1086,Y -24.8979,Z 65,A -46.0797,B 24.8572,C -2.7571,E1 25.1234,E2 129.3073} C_DIS
LIN {X 29.6559,Y -26.6105,Z 65,A -49.2663,B 24.858,C -2.7497,E1 25.1175,E2 132.4972} C_DIS
LIN {X 28.0201,Y -28.3278,Z 65,A -52.6939,B 24.8589,C -2.7413,E1 25.1108,E2 135.9301} C_DIS
LIN {X 26.2016,Y -30.0178,Z 65,A -56.2057,B 24.8596,C -2.7341,E1 25.1035,E2 139.4448} C_DIS
LIN {X 24.3204,Y -31.5612,Z 65,A -59.6363,B 24.8603,C -2.7277,E1 25.096,E2 142.8778} C_DIS
LIN {X 22.5833,Y -32.8272,Z 65,A -62.6667,B 24.8608,C -2.7224,E1 25.0891,E2 145.9101} C_DIS
LIN {X 20.8021,Y -33.9835,Z 65,A -65.8603,B 24.8616,C -2.7146,E1 25.0816,E2 149.112} C_DIS
LIN {X 18.7777,Y -35.1432,Z 65,A -69.1103,B 24.862,C -2.7104,E1 25.0736,E2 152.3624} C_DIS
LIN {X 16.6879,Y -36.1818,Z 65,A -72.3574,B 24.8624,C -2.7068,E1 25.0655,E2 155.6097} C_DIS
LIN {X 14.7997,Y -36.9948,Z 65,A -75.3716,B 24.8629,C -2.7017,E1 25.0577,E2 158.6288} C_DIS
LIN {X 12.7163,Y -37.7609,Z 65,A -78.6001,B 24.8634,C -2.6972,E1 25.0492,E2 161.8615} C_DIS
LIN {X 10.694,Y -38.3831,Z 65,A -81.5103,B 24.8635,C -2.6957,E1 25.0414,E2 164.7701} C_DIS
LIN {X 8.8531,Y -38.8488,Z 65,A -84.2832,B 24.8639,C -2.6925,E1 25.0338,E2 167.5467} C_DIS
LIN {X 6.9039,Y -39.2422,Z 65,A -86.9781,B 24.8639,C -2.6925,E1 25.0264,E2 170.2385} C_DIS
LIN {X 4.9114,Y -39.5413,Z 65,A -90.0224,B 24.8643,C -2.6886,E1 25.018,E2 173.2896} C_DIS
LIN {X 2.8519,Y -39.7427,Z 65,A -93.0373,B 24.8645,C -2.6866,E1 25.0096,E2 176.3076} C_DIS
LIN {X 0.5602,Y -39.841,Z 65,A -96.2591,B 24.8645,C -2.6866,E1 25.0006,E2 179.5287} C_DIS
LIN {X 0.5602,Y -39.841,Z 65,A -96.2591,B 24.8645,C -2.6866,E1 25.0006,E2 179.5287} C_DIS
Enddeposition()
LIN {X 0.2081,Y -41.9548,Z 69.5315,A -96.2626,B 24.8643,C -2.688,E1 25.0006,E2 179.5287} C_DIS
LIN {X 0.2202,Y -48.2941,Z 83.1262,A -96.2298,B 24.8657,C -2.6743,E1 25.0006,E2 179.5287} C_DIS
LIN {X 0.2202,Y -48.2941,Z 104.1262,A -96.5811,B 24.8504,C -2.8219,E1 25.0006,E2 179.5287} C_DIS
LIN {X 0.406,Y -63.8409,Z 104.1262,A -95.3509,B 24.8756,C -2.574,E1 25.0024,E2 178.8883} C_DIS
LIN {X 0.406,Y -63.8409,Z 84.1262,A -95.0165,B 24.8889,C -2.4333,E1 25.0024,E2 178.8883} C_DIS
LIN {X 0.3231,Y -57.5022,Z 70.5315,A -95.0465,B 24.8877,C -2.4459,E1 25.0024,E2 178.8883} C_DIS
LIN {X 0.2954,Y -55.3893,Z 66,A -95.058,B 24.8873,C -2.4508,E1 25.0024,E2 178.8883} C_DIS
Startdeposition()
$VEL.CP = VEL_PRINT
LIN {X 2.8069,Y -55.3215,Z 66,A -92.2608,B 24.8868,C -2.4555,E1 25.0102,E2 176.0805} C_DIS
LIN {X 5.6094,Y -55.1076,Z 66,A -89.3618,B 24.8868,C -2.4568,E1 25.0183,E2 173.1799} C_DIS
LIN {X 8.1554,Y -54.7893,Z 66,A -86.6578,B 24.8865,C -2.4596,E1 25.0258,E2 170.4717} C_DIS
LIN {X 10.8065,Y -54.328,Z 66,A -83.8698,B 24.8862,C -2.4619,E1 25.0335,E2 167.6814} C_DIS
LIN {X 13.4677,Y -53.7299,Z 66,A -81.0641,B 24.886,C -2.4643,E1 25.0411,E2 164.874} C_DIS
LIN {X 16.0795,Y -53.0069,Z 66,A -78.2383,B 24.8857,C -2.4679,E1 25.0487,E2 162.0446} C_DIS
LIN {X 18.7612,Y -52.1187,Z 66,A -75.3122,B 24.8853,C -2.4716,E1 25.0564,E2 159.1155} C_DIS
LIN {X 21.373,Y -51.1028,Z 66,A -72.45,B 24.885,C -2.4748,E1 25.0638,E2 156.2521} C_DIS
LIN {X 23.8526,Y -49.9936,Z 66,A -69.6426,B 24.8846,C -2.4791,E1 25.0709,E2 153.4417} C_DIS
LIN {X 26.3709,Y -48.7121,Z 66,A -66.7279,B 24.8842,C -2.4838,E1 25.0781,E2 150.5241} C_DIS
LIN {X 28.8141,Y -47.3079,Z 66,A -63.8242,B 24.8837,C -2.4888,E1 25.0851,E2 147.6174} C_DIS
LIN {X 31.1971,Y -45.7718,Z 66,A -60.9061,B 24.8832,C -2.4942,E1 25.0919,E2 144.6963} C_DIS
LIN {X 33.5479,Y -44.0783,Z 66,A -57.9439,B 24.8827,C -2.4996,E1 25.0986,E2 141.7319} C_DIS
LIN {X 35.7404,Y -42.3198,Z 66,A -55.0063,B 24.8821,C -2.5066,E1 25.1049,E2 138.789} C_DIS
LIN {X 37.8805,Y -40.4148,Z 66,A -52.0643,B 24.8815,C -2.5129,E1 25.111,E2 135.8438} C_DIS
LIN {X 39.9212,Y -38.4003,Z 66,A -49.1216,B 24.8808,C -2.5195,E1 25.1168,E2 132.8981} C_DIS
LIN {X 41.8542,Y -36.2843,Z 66,A -46.1818,B 24.8802,C -2.5264,E1 25.1222,E2 129.9551} C_DIS
LIN {X 43.6723,Y -34.0753,Z 66,A -43.2156,B 24.8794,C -2.5342,E1 25.1274,E2 126.9843} C_DIS
LIN {X 45.3676,Y -31.7822,Z 66,A -40.2933,B 24.8787,C -2.5415,E1 25.1322,E2 124.0587} C_DIS
LIN {X 46.9361,Y -29.4159,Z 66,A -37.3838,B 24.878,C -2.5491,E1 25.1366,E2 121.146} C_DIS
LIN {X 48.3736,Y -26.9867,Z 66,A -34.5039,B 24.8773,C -2.5565,E1 25.1406,E2 118.2635} C_DIS
LIN {X 49.6894,Y -24.4799,Z 66,A -31.6111,B 24.8766,C -2.5642,E1 25.1443,E2 115.3678} C_DIS
LIN {X 50.8549,Y -21.9568,Z 66,A -28.6669,B 24.8756,C -2.5743,E1 25.1476,E2 112.4157} C_DIS
LIN {X 51.9211,Y -19.2996,Z 66,A -25.8003,B 24.8749,C -2.5811,E1 25.1505,E2 109.549} C_DIS
LIN {X 52.8082,Y -16.7204,Z 66,A -23.0064,B 24.8741,C -2.5891,E1 25.1529,E2 106.752} C_DIS
LIN {X 53.563,Y -14.1176,Z 66,A -20.2138,B 24.8733,C -2.5976,E1 25.155,E2 103.9555} C_DIS
LIN {X 54.2137,Y -11.3671,Z 66,A -17.3472,B 24.8726,C -2.6054,E1 25.1568,E2 101.087} C_DIS
LIN {X 54.6904,Y -8.7956,Z 66,A -14.6076,B 24.8716,C -2.6147,E1 25.1581,E2 98.3415} C_DIS
LIN {X 55.0546,Y -6.1054,Z 66,A -11.8437,B 24.8709,C -2.6225,E1 25.159,E2 95.5754} C_DIS
LIN {X 55.2898,Y -3.3804,Z 66,A -8.9193,B 24.8698,C -2.6336,E1 25.1596,E2 92.6421} C_DIS
LIN {X 55.3883,Y -0.6797,Z 66,A -6.1398,B 24.8689,C -2.6421,E1 25.1598,E2 89.8592} C_DIS
LIN {X 55.3515,Y 2.1334,Z 66,A -3.4257,B 24.8685,C -2.6468,E1 25.1596,E2 87.1501} C_DIS
LIN {X 55.1872,Y 4.7612,Z 66,A -0.6079,B 24.8674,C -2.6574,E1 25.159,E2 84.3238} C_DIS
LIN {X 54.8804,Y 7.5166,Z 66,A 2.1434,B 24.8668,C -2.6637,E1 25.158,E2 81.5739} C_DIS
LIN {X 54.455,Y 10.1477,Z 66,A 4.9309,B 24.8658,C -2.6729,E1 25.1567,E2 78.7812} C_DIS
LIN {X 53.8913,Y 12.8074,Z 66,A 7.7684,B 24.8649,C -2.6819,E1 25.155,E2 75.9386} C_DIS
LIN {X 53.1528,Y 15.5914,Z 66,A 10.6715,B 24.8642,C -2.6891,E1 25.1528,E2 73.0352} C_DIS
LIN {X 52.3272,Y 18.1709,Z 66,A 13.4645,B 24.8634,C -2.6971,E1 25.1503,E2 70.2391} C_DIS
LIN {X 51.3862,Y 20.6832,Z 66,A 16.2308,B 24.8626,C -2.7048,E1 25.1475,E2 67.4699} C_DIS
LIN {X 50.2652,Y 23.2745,Z 66,A 19.1062,B 24.8619,C -2.712,E1 25.1442,E2 64.5932} C_DIS
LIN {X 49.0286,Y 25.7775,Z 66,A 21.9984,B 24.8611,C -2.7199,E1 25.1405,E2 61.6976} C_DIS
LIN {X 47.6714,Y 28.2085,Z 66,A 24.878,B 24.8603,C -2.7275,E1 25.1365,E2 58.815} C_DIS
LIN {X 46.168,Y 30.6075,Z 66,A 27.7885,B 24.8596,C -2.7345,E1 25.1321,E2 55.9025} C_DIS
LIN {X 44.5355,Y 32.9386,Z 66,A 30.7163,B 24.8589,C -2.7413,E1 25.1273,E2 52.9727} C_DIS
LIN {X 42.778,Y 35.1909,Z 66,A 33.68,B 24.8581,C -2.7484,E1 25.1222,E2 50.006} C_DIS
LIN {X 40.9016,Y 37.3545,Z 66,A 36.6216,B 24.8575,C -2.7545,E1 25.1167,E2 47.0631} C_DIS
LIN {X 38.9138,Y 39.4208,Z 66,A 39.5662,B 24.8569,C -2.7603,E1 25.1109,E2 44.1174} C_DIS
LIN {X 36.8224,Y 41.3815,Z 66,A 42.5106,B 24.8563,C -2.7657,E1 25.1048,E2 41.1721} C_DIS
LIN {X 34.6127,Y 43.2473,Z 66,A 45.481,B 24.8558,C -2.7708,E1 25.0984,E2 38.201} C_DIS
LIN {X 32.3627,Y 44.9554,Z 66,A 48.4153,B 24.8552,C -2.776,E1 25.0918,E2 35.2647} C_DIS
LIN {X 30.0137,Y 46.5561,Z 66,A 51.3361,B 24.8548,C -2.7802,E1 25.085,E2 32.3436} C_DIS
LIN {X 27.5993,Y 48.0267,Z 66,A 54.2426,B 24.8544,C -2.7841,E1 25.078,E2 29.4369} C_DIS
LIN {X 25.1047,Y 49.3767,Z 66,A 57.1813,B 24.854,C -2.7879,E1 25.0708,E2 26.4973} C_DIS
LIN {X 22.6427,Y 50.553,Z 66,A 59.9707,B 24.8537,C -2.7905,E1 25.0637,E2 23.709} C_DIS
LIN {X 20.0963,Y 51.6183,Z 66,A 62.8334,B 24.8534,C -2.7935,E1 25.0563,E2 20.8456} C_DIS
LIN {X 17.3756,Y 52.5965,Z 66,A 65.8057,B 24.8532,C -2.7956,E1 25.0485,E2 17.8741} C_DIS
LIN {X 14.7738,Y 53.3855,Z 66,A 68.6026,B 24.853,C -2.7972,E1 25.041,E2 15.0781} C_DIS
LIN {X 12.1365,Y 54.0462,Z 66,A 71.4339,B 24.8528,C -2.7991,E1 25.0333,E2 12.2464} C_DIS
LIN {X 9.4369,Y 54.5832,Z 66,A 74.2515,B 24.8528,C -2.7996,E1 25.0255,E2 9.4308} C_DIS
LIN {X 6.7806,Y 54.9758,Z 66,A 77.0792,B 24.8526,C -2.8012,E1 25.0177,E2 6.6016} C_DIS
LIN {X 4.0588,Y 55.2441,Z 66,A 79.8883,B 24.8526,C -2.801,E1 25.0099,E2 3.7945} C_DIS
LIN {X 1.2295,Y 55.3788,Z 66,A 82.8337,B 24.8526,C -2.801,E1 25.0017,E2 0.8496} C_DIS
LIN {X -1.5642,Y 55.3702,Z 66,A 85.6093,B 24.8529,C -2.7982,E1 24.9939,E2 -1.9193} C_DIS
LIN {X -4.0837,Y 55.2422,Z 66,A 88.4027,B 24.8527,C -2.8007,E1 24.9861,E2 -4.7194} C_DIS
LIN {X -6.8792,Y 54.9638,Z 66,A 91.1557,B 24.8531,C -2.7962,E1 24.9785,E2 -7.4636} C_DIS
LIN {X -9.4787,Y 54.5757,Z 66,A 93.9388,B 24.8531,C -2.7955,E1 24.9708,E2 -10.2476} C_DIS
LIN {X -12.1365,Y 54.0462,Z 66,A 96.7462,B 24.8534,C -2.7933,E1 24.9632,E2 -13.053} C_DIS
LIN {X -14.7822,Y 53.3832,Z 66,A 99.5617,B 24.8537,C -2.7904,E1 24.9556,E2 -15.8658} C_DIS
LIN {X -17.4743,Y 52.5641,Z 66,A 102.4862,B 24.8541,C -2.7873,E1 24.9478,E2 -18.7881} C_DIS
LIN {X -20.0963,Y 51.6183,Z 66,A 105.3873,B 24.8544,C -2.7839,E1 24.9402,E2 -21.6872} C_DIS
LIN {X -22.6427,Y 50.553,Z 66,A 108.2254,B 24.8549,C -2.7795,E1 24.933,E2 -24.5215} C_DIS
LIN {X -25.1047,Y 49.3767,Z 66,A 111.1129,B 24.8552,C -2.7763,E1 24.9257,E2 -27.4088} C_DIS
LIN {X -27.5993,Y 48.0267,Z 66,A 114.0445,B 24.8558,C -2.7712,E1 24.9186,E2 -30.3369} C_DIS
LIN {X -30.0137,Y 46.5561,Z 66,A 116.9803,B 24.8563,C -2.766,E1 24.9117,E2 -33.2697} C_DIS
LIN {X -32.3627,Y 44.9554,Z 66,A 119.9614,B 24.8568,C -2.761,E1 24.9049,E2 -36.2488} C_DIS
LIN {X -34.6358,Y 43.2289,Z 66,A 122.9261,B 24.8574,C -2.755,E1 24.8983,E2 -39.2101} C_DIS
LIN {X -36.8224,Y 41.3815,Z 66,A 125.8964,B 24.8581,C -2.7486,E1 24.8921,E2 -42.1769} C_DIS
LIN {X -38.9138,Y 39.4208,Z 66,A 128.8706,B 24.8588,C -2.7419,E1 24.8861,E2 -45.1473} C_DIS
LIN {X -40.9016,Y 37.3545,Z 66,A 131.845,B 24.8595,C -2.7348,E1 24.8804,E2 -48.1179} C_DIS
LIN {X -42.778,Y 35.1909,Z 66,A 134.8191,B 24.8603,C -2.7275,E1 24.8751,E2 -51.0882} C_DIS
LIN {X -44.5476,Y 32.922,Z 66,A 137.8204,B 24.861,C -2.7201,E1 24.87,E2 -54.0861} C_DIS
LIN {X -46.168,Y 30.6075,Z 66,A 140.7656,B 24.8618,C -2.7126,E1 24.8654,E2 -57.0279} C_DIS
LIN {X -47.6714,Y 28.2085,Z 66,A 143.7044,B 24.8626,C -2.7046,E1 24.8611,E2 -59.9626} C_DIS
LIN {X -49.0286,Y 25.7775,Z 66,A 146.621,B 24.8634,C -2.6969,E1 24.8573,E2 -62.8764} C_DIS
LIN {X -50.2652,Y 23.2745,Z 66,A 149.5189,B 24.8642,C -2.6887,E1 24.8538,E2 -65.7703} C_DIS
LIN {X -51.432,Y 20.5681,Z 66,A 152.5638,B 24.8652,C -2.6795,E1 24.8505,E2 -68.8102} C_DIS
LIN {X -52.382,Y 18.0113,Z 66,A 155.3966,B 24.866,C -2.6711,E1 24.8479,E2 -71.6391} C_DIS
LIN {X -53.2026,Y 15.4193,Z 66,A 158.2169,B 24.8669,C -2.6626,E1 24.8456,E2 -74.4552} C_DIS
LIN {X -53.8953,Y 12.7903,Z 66,A 161.0966,B 24.8676,C -2.655,E1 24.8436,E2 -77.3336} C_DIS
LIN {X -54.468,Y 10.0794,Z 66,A 163.9067,B 24.8686,C -2.6451,E1 24.8421,E2 -80.1367} C_DIS
LIN {X -54.8898,Y 7.4461,Z 66,A 166.7383,B 24.8694,C -2.6377,E1 24.841,E2 -82.9672} C_DIS
LIN {X -55.1879,Y 4.7525,Z 66,A 169.5248,B 24.8703,C -2.6286,E1 24.8402,E2 -85.7487} C_DIS
LIN {X -55.3615,Y 1.8482,Z 66,A 172.4989,B 24.8713,C -2.6185,E1 24.8398,E2 -88.7166} C_DIS
LIN {X -55.385,Y -0.8962,Z 66,A 175.3629,B 24.8721,C -2.61,E1 24.8398,E2 -91.5775} C_DIS
LIN {X -55.2887,Y -3.3967,Z 66,A 178.0839,B 24.8727,C -2.604,E1 24.8402,E2 -94.3006} C_DIS
LIN {X -55.0395,Y -6.2434,Z 66,A -179.0264,B 24.8737,C -2.5938,E1 24.841,E2 -97.1831} C_DIS
LIN {X -54.6897,Y -8.7996,Z 66,A -176.2579,B 24.8743,C -2.5871,E1 24.8422,E2 -99.9524} C_DIS
LIN {X -54.1912,Y -11.4724,Z 66,A -173.4495,B 24.8752,C -2.5785,E1 24.8437,E2 -102.7567} C_DIS
LIN {X -53.5292,Y -14.2463,Z 66,A -170.4605,B 24.876,C -2.5703,E1 24.8457,E2 -105.7435} C_DIS
LIN {X -52.7222,Y -16.9898,Z 66,A -167.5738,B 24.8769,C -2.5605,E1 24.8481,E2 -108.6232} C_DIS
LIN {X -51.8632,Y -19.4557,Z 66,A -164.8142,B 24.8776,C -2.5536,E1 24.8507,E2 -111.3821} C_DIS
LIN {X -50.8549,Y -21.9568,Z 66,A -161.9283,B 24.8782,C -2.5473,E1 24.8538,E2 -114.2691} C_DIS
LIN {X -49.6894,Y -24.4799,Z 66,A -159.0321,B 24.8789,C -2.5398,E1 24.8573,E2 -117.163} C_DIS
LIN {X -48.3513,Y -27.0266,Z 66,A -156.0899,B 24.8797,C -2.5313,E1 24.8612,E2 -120.1005} C_DIS
LIN {X -46.9361,Y -29.4159,Z 66,A -153.1778,B 24.8804,C -2.5246,E1 24.8655,E2 -123.0114} C_DIS
LIN {X -45.3676,Y -31.7822,Z 66,A -150.227,B 24.881,C -2.5176,E1 24.8701,E2 -125.96} C_DIS
LIN {X -43.6689,Y -34.0796,Z 66,A -147.2335,B 24.8816,C -2.5112,E1 24.8752,E2 -128.9526} C_DIS
LIN {X -41.8542,Y -36.2843,Z 66,A -144.2631,B 24.8822,C -2.5048,E1 24.8805,E2 -131.9214} C_DIS
LIN {X -39.9212,Y -38.4003,Z 66,A -141.2907,B 24.8828,C -2.4986,E1 24.8862,E2 -134.8919} C_DIS
LIN {X -37.8805,Y -40.4148,Z 66,A -138.3185,B 24.8834,C -2.4927,E1 24.8922,E2 -137.8624} C_DIS
LIN {X -35.7404,Y -42.3198,Z 66,A -135.3248,B 24.8838,C -2.4876,E1 24.8985,E2 -140.8557} C_DIS
LIN {X -33.5095,Y -44.1077,Z 66,A -132.357,B 24.8843,C -2.4826,E1 24.905,E2 -143.8224} C_DIS
LIN {X -31.1971,Y -45.7718,Z 66,A -129.4086,B 24.8848,C -2.4778,E1 24.9118,E2 -146.7695} C_DIS
LIN {X -28.8141,Y -47.3079,Z 66,A -126.4747,B 24.8852,C -2.4735,E1 24.9187,E2 -149.7024} C_DIS
LIN {X -26.3709,Y -48.7121,Z 66,A -123.5465,B 24.8855,C -2.4699,E1 24.9258,E2 -152.6304} C_DIS
LIN {X -23.8526,Y -49.9936,Z 66,A -120.606,B 24.8858,C -2.4667,E1 24.9332,E2 -155.5711} C_DIS
LIN {X -21.373,Y -51.1028,Z 66,A -117.8235,B 24.8861,C -2.4633,E1 24.9403,E2 -158.352} C_DIS
LIN {X -18.7612,Y -52.1187,Z 66,A -114.8612,B 24.8862,C -2.4619,E1 24.9481,E2 -161.3171} C_DIS
LIN {X -16.0795,Y -53.0069,Z 66,A -111.9977,B 24.8865,C -2.4587,E1 24.9557,E2 -164.1779} C_DIS
LIN {X -13.4592,Y -53.732,Z 66,A -109.1813,B 24.8867,C -2.4571,E1 24.9633,E2 -166.9948} C_DIS
LIN {X -10.7228,Y -54.3449,Z 66,A -106.3146,B 24.8869,C -2.4552,E1 24.9711,E2 -169.8604} C_DIS
LIN {X -8.1191,Y -54.7945,Z 66,A -103.5289,B 24.8869,C -2.4555,E1 24.9788,E2 -172.6493} C_DIS
LIN {X -5.3193,Y -55.1366,Z 66,A -100.6916,B 24.887,C -2.4536,E1 24.9867,E2 -175.4839} C_DIS
LIN {X -2.7092,Y -55.326,Z 66,A -97.8644,B 24.8868,C -2.456,E1 24.9946,E2 -178.3178} C_DIS
LIN {X 0,Y -55.3931,Z 66,A -95.0714,B 24.8868,C -2.4564,E1 25.0024,E2 -181.1117} C_DIS
LIN {X 0,Y -55.3931,Z 66,A -95.0714,B 24.8868,C -2.4564,E1 25.0024,E2 -181.1117} C_DIS
Enddeposition()
LIN {X 0.2833,Y -54.4277,Z 66,A -95.1191,B 24.8858,C -2.4663,E1 25.0024,E2 -181.0876} C_DIS
Startdeposition()
$VEL.CP = VEL_PRINT
LIN {X -1.0024,Y -54.4238,Z 66,A -97.3187,B 24.8874,C -2.4498,E1 24.9961,E2 -178.8488} C_DIS
LIN {X -4.5835,Y -54.2401,Z 66,A -101.2239,B 24.8876,C -2.4472,E1 24.9852,E2 -174.9361} C_DIS
LIN {X -7.0049,Y -53.9804,Z 66,A -103.9065,B 24.8878,C -2.4454,E1 24.9777,E2 -172.2474} C_DIS
LIN {X -9.6214,Y -53.576,Z 66,A -106.9217,B 24.8881,C -2.442,E1 24.9694,E2 -169.2214} C_DIS
LIN {X -13.7924,Y -52.6568,Z 66,A -110.8274,B 24.8869,C -2.4549,E1 24.9588,E2 -165.3413} C_DIS
LIN {X -15.7918,Y -52.0919,Z 66,A -114.5617,B 24.8893,C -2.4289,E1 24.9487,E2 -161.5387} C_DIS
LIN {X -19.2852,Y -50.9022,Z 66,A -116.7374,B 24.8862,C -2.4624,E1 24.9432,E2 -159.4383} C_DIS
LIN {X -22.1332,Y -49.7299,Z 66,A -120.5449,B 24.8868,C -2.4557,E1 24.9333,E2 -155.6061} C_DIS
LIN {X -24.7475,Y -48.4821,Z 66,A -123.5695,B 24.8864,C -2.4597,E1 24.9257,E2 -152.5832} C_DIS
LIN {X -27.1963,Y -47.1521,Z 66,A -126.4876,B 24.8861,C -2.4639,E1 24.9186,E2 -149.6667} C_DIS
LIN {X -29.4735,Y -45.7633,Z 66,A -129.3481,B 24.8858,C -2.4672,E1 24.9118,E2 -146.8049} C_DIS
LIN {X -32.1624,Y -43.9151,Z 66,A -132.5305,B 24.8848,C -2.477,E1 24.9046,E2 -143.6351} C_DIS
LIN {X -34.0481,Y -42.4708,Z 66,A -135.3366,B 24.8849,C -2.4763,E1 24.8984,E2 -140.8168} C_DIS
LIN {X -36.1743,Y -40.6744,Z 66,A -138.2758,B 24.8844,C -2.4817,E1 24.8922,E2 -137.879} C_DIS
LIN {X -38.2494,Y -38.7291,Z 66,A -141.2935,B 24.8839,C -2.4873,E1 24.8861,E2 -134.8623} C_DIS
LIN {X -39.8498,Y -37.0814,Z 66,A -143.7148,B 24.8834,C -2.4924,E1 24.8815,E2 -132.4426} C_DIS
LIN {X -41.8395,Y -34.8197,Z 66,A -146.5343,B 24.8822,C -2.5053,E1 24.8764,E2 -129.6409} C_DIS
LIN {X -43.0989,Y -33.2481,Z 66,A -149.0477,B 24.8823,C -2.5038,E1 24.872,E2 -127.1123} C_DIS
LIN {X -44.7894,Y -30.9336,Z 66,A -152.069,B 24.8816,C -2.5111,E1 24.8671,E2 -124.0936} C_DIS
LIN {X -46.3701,Y -28.51,Z 66,A -155.1202,B 24.8809,C -2.5188,E1 24.8626,E2 -121.0452} C_DIS
LIN {X -48.1356,Y -25.415,Z 66,A -158.4757,B 24.8794,C -2.535,E1 24.858,E2 -117.7108} C_DIS
LIN {X -49.2715,Y -23.1352,Z 66,A -161.5249,B 24.8792,C -2.5365,E1 24.8543,E2 -114.6487} C_DIS
LIN {X -50.2599,Y -20.9018,Z 66,A -164.0929,B 24.8785,C -2.5437,E1 24.8514,E2 -112.0838} C_DIS
LIN {X -51.2485,Y -18.3459,Z 66,A -167.0047,B 24.8778,C -2.5516,E1 24.8486,E2 -109.1743} C_DIS
LIN {X -52.095,Y -15.7816,Z 66,A -169.872,B 24.877,C -2.5595,E1 24.8462,E2 -106.3096} C_DIS
LIN {X -52.8054,Y -13.2112,Z 66,A -172.9486,B 24.8766,C -2.5638,E1 24.844,E2 -103.2252} C_DIS
LIN {X -53.4044,Y -10.5348,Z 66,A -175.4261,B 24.8751,C -2.5788,E1 24.8426,E2 -100.769} C_DIS
LIN {X -53.8014,Y -8.2685,Z 66,A -178.1129,B 24.8748,C -2.5822,E1 24.8414,E2 -98.0744} C_DIS
LIN {X -54.1571,Y -5.4758,Z 66,A 178.9315,B 24.8739,C -2.5915,E1 24.8404,E2 -95.1233} C_DIS
LIN {X -54.3649,Y -2.7306,Z 66,A 175.7902,B 24.8734,C -2.5968,E1 24.8399,E2 -91.9759} C_DIS
LIN {X -54.4304,Y 0.5692,Z 66,A 172.6001,B 24.8719,C -2.6121,E1 24.8399,E2 -88.803} C_DIS
LIN {X -54.3528,Y 2.9555,Z 66,A 169.9471,B 24.8713,C -2.6178,E1 24.8401,E2 -86.1479} C_DIS
LIN {X -54.1369,Y 5.6705,Z 66,A 167.0665,B 24.8705,C -2.6267,E1 24.8409,E2 -83.2711} C_DIS
LIN {X -53.7639,Y 8.5111,Z 66,A 164.1328,B 24.8694,C -2.6374,E1 24.842,E2 -80.3455} C_DIS
LIN {X -53.427,Y 10.4177,Z 66,A 161.9398,B 24.869,C -2.6414,E1 24.8432,E2 -78.1491} C_DIS
LIN {X -52.8529,Y 13.0208,Z 66,A 159.1526,B 24.8681,C -2.6504,E1 24.8449,E2 -75.3672} C_DIS
LIN {X -52.1321,Y 15.6589,Z 66,A 156.3004,B 24.8672,C -2.6597,E1 24.8471,E2 -72.5206} C_DIS
LIN {X -51.1144,Y 18.7157,Z 66,A 152.8155,B 24.8663,C -2.6685,E1 24.8503,E2 -69.0371} C_DIS
LIN {X -50.053,Y 21.3931,Z 66,A 149.4051,B 24.866,C -2.6718,E1 24.854,E2 -65.6155} C_DIS
LIN {X -48.3524,Y 25.0014,Z 66,A 145.8783,B 24.8637,C -2.6944,E1 24.8582,E2 -62.1236} C_DIS
LIN {X -46.9206,Y 27.5939,Z 66,A 142.3408,B 24.8634,C -2.6967,E1 24.8631,E2 -58.5731} C_DIS
LIN {X -45.4243,Y 29.9932,Z 66,A 139.4134,B 24.8625,C -2.7056,E1 24.8675,E2 -55.6524} C_DIS
LIN {X -43.5661,Y 32.6336,Z 66,A 136.1519,B 24.8614,C -2.7169,E1 24.8728,E2 -52.4017} C_DIS
LIN {X -41.9983,Y 34.6287,Z 66,A 133.3003,B 24.861,C -2.7209,E1 24.8778,E2 -49.5464} C_DIS
LIN {X -40.1351,Y 36.7714,Z 66,A 130.2793,B 24.8603,C -2.7278,E1 24.8834,E2 -46.5284} C_DIS
LIN {X -37.9327,Y 39.0398,Z 66,A 126.9751,B 24.8594,C -2.736,E1 24.8899,E2 -43.2299} C_DIS
LIN {X -36.273,Y 40.586,Z 66,A 124.5402,B 24.8589,C -2.7407,E1 24.895,E2 -40.7963} C_DIS
LIN {X -34.0871,Y 42.4392,Z 66,A 121.5486,B 24.8582,C -2.7476,E1 24.9014,E2 -37.8098} C_DIS
LIN {X -31.9633,Y 44.0609,Z 66,A 118.711,B 24.8577,C -2.7529,E1 24.9077,E2 -34.9747} C_DIS
LIN {X -29.5385,Y 45.7213,Z 66,A 115.2545,B 24.8577,C -2.7529,E1 24.9158,E2 -31.5067} C_DIS
LIN {X -26.6309,Y 47.4738,Z 66,A 112.0033,B 24.8565,C -2.7644,E1 24.9236,E2 -28.2734} C_DIS
LIN {X -24.1514,Y 48.7818,Z 66,A 109.0465,B 24.856,C -2.769,E1 24.931,E2 -25.3197} C_DIS
LIN {X -19.9206,Y 50.657,Z 66,A 104.3349,B 24.855,C -2.7787,E1 24.943,E2 -20.62} C_DIS
LIN {X -17.304,Y 51.6094,Z 66,A 101.6935,B 24.8541,C -2.7873,E1 24.9499,E2 -17.9939} C_DIS
LIN {X -15.5915,Y 52.1524,Z 66,A 99.2748,B 24.8548,C -2.7802,E1 24.9564,E2 -15.5543} C_DIS
LIN {X -12.7507,Y 52.9188,Z 66,A 96.2556,B 24.8544,C -2.7846,E1 24.9646,E2 -12.541} C_DIS
LIN {X -10.0639,Y 53.4947,Z 66,A 93.3578,B 24.8541,C -2.7868,E1 24.9725,E2 -9.6453} C_DIS
LIN {X -7.0054,Y 53.9804,Z 66,A 90.2628,B 24.8536,C -2.7919,E1 24.981,E2 -6.5597} C_DIS
LIN {X -4.6037,Y 54.2382,Z 66,A 87.4413,B 24.854,C -2.7882,E1 24.9889,E2 -3.7278} C_DIS
LIN {X -1.7567,Y 54.4048,Z 66,A 84.6684,B 24.8534,C -2.7933,E1 24.9966,E2 -0.9666} C_DIS
LIN {X 0.603,Y 54.4303,Z 66,A 81.9729,B 24.8538,C -2.7899,E1 25.0041,E2 1.7369} C_DIS
LIN {X 3.4712,Y 54.3225,Z 66,A 78.2957,B 24.855,C -2.778,E1 25.0145,E2 5.441} C_DIS
LIN {X 7.4824,Y 53.9166,Z 66,A 74.6312,B 24.854,C -2.7879,E1 25.0246,E2 9.0792} C_DIS
LIN {X 10.8717,Y 53.3364,Z 66,A 71.4469,B 24.8533,C -2.7947,E1 25.0333,E2 12.2438} C_DIS
LIN {X 14.0991,Y 52.5755,Z 66,A 67.1654,B 24.8551,C -2.7778,E1 25.0449,E2 16.5592} C_DIS
LIN {X 17.6942,Y 51.4768,Z 66,A 63.7111,B 24.8544,C -2.7843,E1 25.0541,E2 19.9916} C_DIS
LIN {X 20.3453,Y 50.4882,Z 66,A 60.7009,B 24.8547,C -2.7808,E1 25.0619,E2 23.0035} C_DIS
LIN {X 22.8734,Y 49.394,Z 66,A 57.9039,B 24.8549,C -2.7796,E1 25.069,E2 25.7964} C_DIS
LIN {X 24.5359,Y 48.5896,Z 66,A 55.9058,B 24.8552,C -2.7762,E1 25.074,E2 27.7972} C_DIS
LIN {X 26.9905,Y 47.2704,Z 66,A 53.0005,B 24.8556,C -2.7727,E1 25.0811,E2 30.7021} C_DIS
LIN {X 29.5149,Y 45.7367,Z 66,A 50.2235,B 24.8554,C -2.7748,E1 25.0877,E2 33.4656} C_DIS
LIN {X 30.828,Y 44.8629,Z 66,A 48.172,B 24.8565,C -2.7642,E1 25.0925,E2 35.5352} C_DIS
LIN {X 33.1712,Y 43.1582,Z 66,A 45.1417,B 24.857,C -2.7594,E1 25.0992,E2 38.566} C_DIS
LIN {X 35.3374,Y 41.4032,Z 66,A 42.2549,B 24.8575,C -2.7549,E1 25.1054,E2 41.4524} C_DIS
LIN {X 37.4708,Y 39.4836,Z 66,A 39.2293,B 24.8581,C -2.7488,E1 25.1116,E2 44.4802} C_DIS
LIN {X 39.4241,Y 37.5331,Z 66,A 36.4526,B 24.8584,C -2.7453,E1 25.1171,E2 47.2532} C_DIS
LIN {X 41.0075,Y 35.7958,Z 66,A 33.9596,B 24.8591,C -2.7394,E1 25.1217,E2 49.749} C_DIS
LIN {X 42.5708,Y 33.9224,Z 66,A 31.4697,B 24.8595,C -2.7351,E1 25.1261,E2 52.2376} C_DIS
LIN {X 44.1446,Y 31.8474,Z 66,A 28.6238,B 24.8604,C -2.7263,E1 25.1308,E2 55.0906} C_DIS
LIN {X 45.7777,Y 29.4509,Z 66,A 25.5528,B 24.8612,C -2.7183,E1 25.1356,E2 58.1654} C_DIS
LIN {X 47.2639,Y 27.0019,Z 66,A 22.5722,B 24.862,C -2.7112,E1 25.1398,E2 61.1475} C_DIS
LIN {X 48.5763,Y 24.5623,Z 66,A 19.7471,B 24.8626,C -2.7052,E1 25.1435,E2 63.9717} C_DIS
LIN {X 49.8229,Y 21.9239,Z 66,A 16.9306,B 24.8629,C -2.7022,E1 25.1467,E2 66.7802} C_DIS
LIN {X 50.6663,Y 19.8967,Z 66,A 14.3029,B 24.8642,C -2.6888,E1 25.1495,E2 69.425} C_DIS
LIN {X 51.6552,Y 17.1672,Z 66,A 11.091,B 24.8655,C -2.6766,E1 25.1525,E2 72.6478} C_DIS
LIN {X 52.4487,Y 14.5631,Z 66,A 8.4498,B 24.8658,C -2.6729,E1 25.1545,E2 75.2825} C_DIS
LIN {X 53.1228,Y 11.872,Z 66,A 5.5308,B 24.8667,C -2.6641,E1 25.1564,E2 78.2053} C_DIS
LIN {X 53.6679,Y 9.0954,Z 66,A 2.166,B 24.8685,C -2.6467,E1 25.158,E2 81.5917} C_DIS
LIN {X 54.2034,Y 4.995,Z 66,A -1.2892,B 24.8679,C -2.6527,E1 25.1592,E2 85.0123} C_DIS
LIN {X 54.349,Y 3.0236,Z 66,A -3.8311,B 24.8695,C -2.6361,E1 25.1596,E2 87.5783} C_DIS
LIN {X 54.4314,Y 0.0761,Z 66,A -6.4268,B 24.8694,C -2.6375,E1 25.1598,E2 90.1553} C_DIS
LIN {X 54.3654,Y -2.707,Z 66,A -10.2748,B 24.8723,C -2.6082,E1 25.1594,E2 94.0497} C_DIS
LIN {X 54.1443,Y -5.5997,Z 66,A -13.245,B 24.873,C -2.6003,E1 25.1586,E2 97.0208} C_DIS
LIN {X 53.5284,Y -9.8851,Z 66,A -17.2431,B 24.8733,C -2.5982,E1 25.1568,E2 101.0005} C_DIS
LIN {X 52.6558,Y -13.796,Z 66,A -22.2028,B 24.8761,C -2.569,E1 25.1535,E2 106.0006} C_DIS
LIN {X 51.3352,Y -18.1006,Z 66,A -26.3021,B 24.8761,C -2.5683,E1 25.15,E2 110.0782} C_DIS
LIN {X 50.3061,Y -20.7906,Z 66,A -29.1925,B 24.8768,C -2.5622,E1 25.147,E2 112.9671} C_DIS
LIN {X 49.2447,Y -23.1935,Z 66,A -32.163,B 24.878,C -2.5496,E1 25.1436,E2 115.9513} C_DIS
LIN {X 48.0343,Y -25.6074,Z 66,A -34.8031,B 24.8783,C -2.5457,E1 25.1402,E2 118.5866} C_DIS
LIN {X 46.7261,Y -27.9228,Z 66,A -37.6405,B 24.8792,C -2.537,E1 25.1362,E2 121.4301} C_DIS
LIN {X 45.1805,Y -30.3598,Z 66,A -40.703,B 24.88,C -2.5281,E1 25.1315,E2 124.4983} C_DIS
LIN {X 43.4869,Y -32.739,Z 66,A -43.6998,B 24.8807,C -2.5215,E1 25.1265,E2 127.4962} C_DIS
LIN {X 41.737,Y -34.943,Z 66,A -46.6053,B 24.8813,C -2.515,E1 25.1214,E2 130.4035} C_DIS
LIN {X 39.9309,Y -36.9936,Z 66,A -49.4618,B 24.8819,C -2.5083,E1 25.1161,E2 133.2633} C_DIS
LIN {X 38.0175,Y -38.9577,Z 66,A -52.3167,B 24.8825,C -2.5021,E1 25.1104,E2 136.1209} C_DIS
LIN {X 35.9891,Y -40.8387,Z 66,A -55.2401,B 24.8831,C -2.4952,E1 25.1044,E2 139.0488} C_DIS
LIN {X 33.9187,Y -42.5737,Z 66,A -58.0796,B 24.8837,C -2.4891,E1 25.0982,E2 141.8919} C_DIS
LIN {X 31.7781,Y -44.1944,Z 66,A -60.9166,B 24.8843,C -2.4831,E1 25.0918,E2 144.733} C_DIS
LIN {X 29.4915,Y -45.7517,Z 66,A -63.6409,B 24.8844,C -2.4813,E1 25.0855,E2 147.4525} C_DIS
LIN {X 27.462,Y -46.9986,Z 66,A -66.2796,B 24.8851,C -2.4741,E1 25.0792,E2 150.1002} C_DIS
LIN {X 25.0332,Y -48.3357,Z 66,A -69.2243,B 24.8856,C -2.4686,E1 25.0719,E2 153.0494} C_DIS
LIN {X 22.6761,Y -49.4848,Z 66,A -71.9993,B 24.886,C -2.464,E1 25.0649,E2 155.8281} C_DIS
LIN {X 20.051,Y -50.6056,Z 66,A -74.9684,B 24.8864,C -2.4605,E1 25.0572,E2 158.7988} C_DIS
LIN {X 17.4025,Y -51.5763,Z 66,A -77.7727,B 24.8864,C -2.46,E1 25.0499,E2 161.5984} C_DIS
LIN {X 15.6042,Y -52.1485,Z 66,A -80.5437,B 24.8881,C -2.4423,E1 25.0424,E2 164.4066} C_DIS
LIN {X 10.2383,Y -53.4615,Z 66,A -86.5037,B 24.8888,C -2.4344,E1 25.0261,E2 170.3777} C_DIS
LIN {X 4.4499,Y -54.251,Z 66,A -91.6973,B 24.8874,C -2.449,E1 25.0118,E2 175.5326} C_DIS
LIN {X 1.5073,Y -54.4122,Z 66,A -95.0635,B 24.888,C -2.4429,E1 25.0023,E2 178.9124} C_DIS
LIN {X 1.5073,Y -54.4122,Z 66,A -95.0635,B 24.888,C -2.4429,E1 25.0023,E2 178.9124} C_DIS
Enddeposition()
LIN {X 0.2758,Y -53.4677,Z 66,A -95.4254,B 24.8848,C -2.477,E1 25.0016,E2 179.1932} C_DIS
Startdeposition()
$VEL.CP = VEL_PRINT
LIN {X 3.0149,Y -53.3888,Z 66,A -92.1695,B 24.8842,C -2.484,E1 25.0107,E2 175.9215} C_DIS
LIN {X 4.8149,Y -53.2567,Z 66,A -90.3219,B 24.8842,C -2.4833,E1 25.0158,E2 174.0766} C_DIS
LIN {X 7.4129,Y -52.9578,Z 66,A -86.8997,B 24.883,C -2.4971,E1 25.0254,E2 170.6245} C_DIS
LIN {X 10.4297,Y -52.4472,Z 66,A -83.4264,B 24.8823,C -2.5036,E1 25.0349,E2 167.1397} C_DIS
LIN {X 14.8976,Y -51.3567,Z 66,A -79.2956,B 24.8834,C -2.4927,E1 25.046,E2 163.0409} C_DIS
LIN {X 16.5574,Y -50.846,Z 66,A -76.4157,B 24.8812,C -2.5154,E1 25.0538,E2 160.1128} C_DIS
LIN {X 20.5103,Y -49.384,Z 66,A -72.6509,B 24.8821,C -2.5063,E1 25.0635,E2 156.3778} C_DIS
LIN {X 23.0129,Y -48.2689,Z 66,A -69.7339,B 24.8817,C -2.5104,E1 25.0709,E2 153.4585} C_DIS
LIN {X 25.5127,Y -46.9954,Z 66,A -66.7402,B 24.8813,C -2.5152,E1 25.0783,E2 150.462} C_DIS
LIN {X 27.0437,Y -46.1318,Z 66,A -64.3934,B 24.88,C -2.5281,E1 25.084,E2 148.0917} C_DIS
LIN {X 30.4321,Y -43.9701,Z 66,A -60.5387,B 24.8801,C -2.527,E1 25.0929,E2 144.2524} C_DIS
LIN {X 32.7324,Y -42.2856,Z 66,A -57.5325,B 24.8796,C -2.5323,E1 25.0996,E2 141.2444} C_DIS
LIN {X 34.8556,Y -40.5538,Z 66,A -54.579,B 24.879,C -2.5392,E1 25.106,E2 138.2862} C_DIS
LIN {X 36.26,Y -39.3027,Z 66,A -52.5232,B 24.8784,C -2.5446,E1 25.1102,E2 136.2257} C_DIS
LIN {X 38.7141,Y -36.8881,Z 66,A -48.9106,B 24.8778,C -2.5519,E1 25.1173,E2 132.6114} C_DIS
LIN {X 40.5688,Y -34.838,Z 66,A -45.9758,B 24.8771,C -2.5587,E1 25.1227,E2 129.6736} C_DIS
LIN {X 42.2868,Y -32.7308,Z 66,A -43.3671,B 24.877,C -2.5598,E1 25.1273,E2 127.0745} C_DIS
LIN {X 43.7351,Y -30.7693,Z 66,A -39.8856,B 24.8745,C -2.5856,E1 25.133,E2 123.549} C_DIS
LIN {X 45.9146,Y -27.411,Z 66,A -36.2189,B 24.8746,C -2.584,E1 25.1384,E2 119.9045} C_DIS
LIN {X 47.27,Y -25.0005,Z 66,A -33.7527,B 24.8749,C -2.5818,E1 25.1417,E2 117.4564} C_DIS
LIN {X 49.0017,Y -21.408,Z 66,A -29.3004,B 24.8733,C -2.5982,E1 25.147,E2 112.9893} C_DIS
LIN {X 49.7118,Y -19.702,Z 66,A -27.107,B 24.8722,C -2.6088,E1 25.1493,E2 110.7831} C_DIS
LIN {X 50.5965,Y -17.3047,Z 66,A -24.6146,B 24.8719,C -2.6117,E1 25.1516,E2 108.2976} C_DIS
LIN {X 51.1117,Y -15.7176,Z 66,A -22.1311,B 24.8699,C -2.6325,E1 25.1537,E2 105.7792} C_DIS
LIN {X 52.2773,Y -11.2493,Z 66,A -17.8733,B 24.8699,C -2.6327,E1 25.1565,E2 101.5455} C_DIS
LIN {X 52.8334,Y -8.2526,Z 66,A -14.0817,B 24.8677,C -2.6545,E1 25.1583,E2 97.7246} C_DIS
LIN {X 53.2437,Y -4.9579,Z 66,A -11.1692,B 24.868,C -2.6516,E1 25.1592,E2 94.8363} C_DIS
LIN {X 53.4208,Y -2.3843,Z 66,A -7.9749,B 24.8662,C -2.6697,E1 25.1597,E2 91.6181} C_DIS
LIN {X 53.4717,Y 0.3702,Z 66,A -4.4901,B 24.864,C -2.6907,E1 25.1597,E2 88.1042} C_DIS
LIN {X 53.3185,Y 4.0779,Z 66,A -0.9143,B 24.8637,C -2.6943,E1 25.1591,E2 84.5412} C_DIS
LIN {X 52.8911,Y 7.8792,Z 66,A 2.5111,B 24.8639,C -2.6923,E1 25.1579,E2 81.1408} C_DIS
LIN {X 52.42,Y 10.5652,Z 66,A 6.1986,B 24.8613,C -2.7179,E1 25.1559,E2 77.4143} C_DIS
LIN {X 51.3979,Y 14.7555,Z 66,A 10.5401,B 24.8605,C -2.7256,E1 25.1528,E2 73.0796} C_DIS
LIN {X 50.3207,Y 18.0926,Z 66,A 14.059,B 24.8599,C -2.7314,E1 25.1497,E2 69.5668} C_DIS
LIN {X 49.3963,Y 20.4807,Z 66,A 16.8416,B 24.859,C -2.74,E1 25.1467,E2 66.7792} C_DIS
LIN {X 47.8136,Y 23.9451,Z 66,A 20.8479,B 24.858,C -2.7496,E1 25.1419,E2 62.7717} C_DIS
LIN {X 46.4713,Y 26.4562,Z 66,A 23.8684,B 24.8572,C -2.7571,E1 25.1379,E2 59.7493} C_DIS
LIN {X 45.3487,Y 28.3366,Z 66,A 26.5618,B 24.8558,C -2.7705,E1 25.1339,E2 57.0378} C_DIS
LIN {X 43.2591,Y 31.435,Z 66,A 30.1936,B 24.8556,C -2.7725,E1 25.1281,E2 53.4192} C_DIS
LIN {X 41.8887,Y 33.2388,Z 66,A 33.0996,B 24.854,C -2.7882,E1 25.123,E2 50.4894} C_DIS
LIN {X 39.5667,Y 35.9723,Z 66,A 36.3815,B 24.8543,C -2.7851,E1 25.117,E2 47.2298} C_DIS
LIN {X 37.0643,Y 38.5449,Z 66,A 39.9362,B 24.8541,C -2.7871,E1 25.11,E2 43.6854} C_DIS
LIN {X 35.0355,Y 40.3982,Z 66,A 43.1628,B 24.8529,C -2.7986,E1 25.1033,E2 40.4444} C_DIS
LIN {X 32.9032,Y 42.1538,Z 66,A 46.1202,B 24.8523,C -2.8039,E1 25.0968,E2 37.4855} C_DIS
LIN {X 30.7395,Y 43.7563,Z 66,A 48.8294,B 24.8522,C -2.8052,E1 25.0907,E2 34.7828} C_DIS
LIN {X 28.7172,Y 45.1091,Z 66,A 52.3017,B 24.8499,C -2.8267,E1 25.0825,E2 31.2708} C_DIS
LIN {X 25.0786,Y 47.2289,Z 66,A 55.8282,B 24.8513,C -2.8131,E1 25.074,E2 27.7869} C_DIS
LIN {X 22.0606,Y 48.7114,Z 66,A 59.8317,B 24.85,C -2.8252,E1 25.0639,E2 23.7651} C_DIS
LIN {X 19.3067,Y 49.867,Z 66,A 62.9098,B 24.85,C -2.826,E1 25.0559,E2 20.692} C_DIS
LIN {X 16.5814,Y 50.8384,Z 66,A 65.5106,B 24.8507,C -2.819,E1 25.0491,E2 18.1131} C_DIS
LIN {X 13.8736,Y 51.6429,Z 66,A 69.4053,B 24.8487,C -2.8377,E1 25.0385,E2 14.1806} C_DIS
LIN {X 10.7647,Y 52.3793,Z 66,A 71.9805,B 24.8503,C -2.8233,E1 25.0316,E2 11.643} C_DIS
LIN {X 8.2099,Y 52.84,Z 66,A 75.3565,B 24.849,C -2.8353,E1 25.0222,E2 8.2419} C_DIS
LIN {X 4.8354,Y 53.2546,Z 66,A 79.1517,B 24.8486,C -2.8387,E1 25.0117,E2 4.4413} C_DIS
LIN {X 1.6859,Y 53.4474,Z 66,A 81.881,B 24.8499,C -2.8265,E1 25.0042,E2 1.7417} C_DIS
LIN {X -0.4748,Y 53.472,Z 66,A 84.4865,B 24.8494,C -2.8314,E1 24.9969,E2 -0.8752} C_DIS
LIN {X -2.7894,Y 53.4014,Z 66,A 86.8437,B 24.8497,C -2.8283,E1 24.9903,E2 -3.2256} C_DIS
LIN {X -5.5626,Y 53.1839,Z 66,A 89.9224,B 24.8497,C -2.8287,E1 24.9817,E2 -6.3066} C_DIS
LIN {X -9.9711,Y 52.5361,Z 66,A 94.7788,B 24.8499,C -2.8268,E1 24.9683,E2 -11.1631} C_DIS
LIN {X -12.7421,Y 51.9337,Z 66,A 97.8474,B 24.8501,C -2.8246,E1 24.96,E2 -14.2304} C_DIS
LIN {X -15.508,Y 51.1758,Z 66,A 100.7756,B 24.8507,C -2.8189,E1 24.9522,E2 -17.1497} C_DIS
LIN {X -19.3185,Y 49.8624,Z 66,A 104.9569,B 24.8515,C -2.8112,E1 24.9412,E2 -21.3209} C_DIS
LIN {X -21.3369,Y 49.032,Z 66,A 107.3427,B 24.8518,C -2.8087,E1 24.935,E2 -23.7063} C_DIS
LIN {X -24.0141,Y 47.7781,Z 66,A 111.2667,B 24.851,C -2.8166,E1 24.9251,E2 -27.6592} C_DIS
LIN {X -26.7785,Y 46.2861,Z 66,A 114.4257,B 24.852,C -2.8073,E1 24.9175,E2 -30.8053} C_DIS
LIN {X -29.8032,Y 44.3988,Z 66,A 117.7422,B 24.8536,C -2.7918,E1 24.9098,E2 -34.0956} C_DIS
LIN {X -31.8372,Y 42.9641,Z 66,A 120.6642,B 24.8537,C -2.7907,E1 24.9031,E2 -37.025} C_DIS
LIN {X -34.0433,Y 41.2377,Z 66,A 123.7057,B 24.8543,C -2.7849,E1 24.8965,E2 -40.0642} C_DIS
LIN {X -35.7382,Y 39.7776,Z 66,A 126.1576,B 24.8548,C -2.7805,E1 24.8914,E2 -42.5153} C_DIS
LIN {X -37.7221,Y 37.9016,Z 66,A 128.8823,B 24.8558,C -2.7704,E1 24.886,E2 -45.2274} C_DIS
LIN {X -39.3656,Y 36.1914,Z 66,A 131.6023,B 24.8562,C -2.7671,E1 24.8808,E2 -47.9513} C_DIS
LIN {X -41.198,Y 34.0911,Z 66,A 134.5889,B 24.857,C -2.7596,E1 24.8754,E2 -50.9335} C_DIS
LIN {X -42.4774,Y 32.4836,Z 66,A 137.0733,B 24.857,C -2.7583,E1 24.8711,E2 -53.4268} C_DIS
LIN {X -44.6198,Y 29.4709,Z 66,A 140.5038,B 24.8591,C -2.7393,E1 24.8657,E2 -56.8287} C_DIS
LIN {X -45.9168,Y 27.4055,Z 66,A 143.9387,B 24.8585,C -2.7449,E1 24.8607,E2 -60.2946} C_DIS
LIN {X -47.548,Y 24.4679,Z 66,A 147.0586,B 24.8603,C -2.727,E1 24.8566,E2 -63.3883} C_DIS
LIN {X -48.7144,Y 22.0537,Z 66,A 150.3588,B 24.8605,C -2.7253,E1 24.8528,E2 -66.7023} C_DIS
LIN {X -49.9971,Y 18.9673,Z 66,A 154.5947,B 24.8605,C -2.7247,E1 24.8485,E2 -70.9607} C_DIS
LIN {X -51.1059,Y 15.7373,Z 66,A 157.2125,B 24.8634,C -2.6973,E1 24.8463,E2 -73.528} C_DIS
LIN {X -51.8476,Y 13.0876,Z 66,A 160.2162,B 24.8642,C -2.6891,E1 24.8442,E2 -76.5295} C_DIS
LIN {X -52.3558,Y 10.8791,Z 66,A 163.135,B 24.8642,C -2.6891,E1 24.8425,E2 -79.4654} C_DIS
LIN {X -53.0125,Y 7.0109,Z 66,A 166.9129,B 24.8662,C -2.6693,E1 24.8409,E2 -83.2186} C_DIS
LIN {X -53.3128,Y 4.1499,Z 66,A 169.9673,B 24.8672,C -2.6592,E1 24.8401,E2 -86.267} C_DIS
LIN {X -53.4574,Y 1.3326,Z 66,A 173.0227,B 24.8681,C -2.6502,E1 24.8398,E2 -89.3193} C_DIS
LIN {X -53.4042,Y -2.7399,Z 66,A 177.3086,B 24.8696,C -2.6353,E1 24.8401,E2 -93.5954} C_DIS
LIN {X -53.2066,Y -5.3421,Z 66,A -179.7259,B 24.8702,C -2.6292,E1 24.8408,E2 -96.5641} C_DIS
LIN {X -52.8792,Y -7.9566,Z 66,A -176.8991,B 24.8711,C -2.6205,E1 24.8419,E2 -99.3871} C_DIS
LIN {X -52.2679,Y -11.2932,Z 66,A -172.3843,B 24.8708,C -2.6232,E1 24.8445,E2 -103.935} C_DIS
LIN {X -51.1483,Y -15.5988,Z 66,A -168.5107,B 24.8736,C -2.595,E1 24.8474,E2 -107.7637} C_DIS
LIN {X -50.5017,Y -17.5802,Z 66,A -165.343,B 24.8728,C -2.6033,E1 24.8503,E2 -110.9691} C_DIS
LIN {X -49.0898,Y -21.2059,Z 66,A -161.9138,B 24.8751,C -2.5797,E1 24.8539,E2 -114.3611} C_DIS
LIN {X -47.4614,Y -24.6355,Z 66,A -158.3711,B 24.8769,C -2.5603,E1 24.8582,E2 -117.8765} C_DIS
LIN {X -46.3065,Y -26.7428,Z 66,A -155.6327,B 24.8773,C -2.5561,E1 24.862,E2 -120.6192} C_DIS
LIN {X -45.0292,Y -28.8417,Z 66,A -152.6477,B 24.8774,C -2.555,E1 24.8664,E2 -123.6168} C_DIS
LIN {X -43.4572,Y -31.1602,Z 66,A -149.6469,B 24.8782,C -2.5476,E1 24.8712,E2 -126.6148} C_DIS
LIN {X -42.0649,Y -33.0158,Z 66,A -146.6818,B 24.878,C -2.5496,E1 24.8763,E2 -129.5987} C_DIS
LIN {X -39.619,Y -35.9148,Z 66,A -143.2356,B 24.8798,C -2.5304,E1 24.8826,E2 -133.0146} C_DIS
LIN {X -38.2388,Y -37.3803,Z 66,A -140.4053,B 24.8792,C -2.5371,E1 24.8881,E2 -135.873} C_DIS
LIN {X -35.5816,Y -39.9178,Z 66,A -136.9547,B 24.8807,C -2.5212,E1 24.8952,E2 -139.2996} C_DIS
LIN {X -33.4381,Y -41.7307,Z 66,A -134.1013,B 24.8815,C -2.513,E1 24.9013,E2 -142.1445} C_DIS
LIN {X -31.2285,Y -43.4083,Z 66,A -130.8172,B 24.8815,C -2.5133,E1 24.9087,E2 -145.4408} C_DIS
LIN {X -28.0643,Y -45.5183,Z 66,A -127.2626,B 24.8829,C -2.4982,E1 24.917,E2 -148.9708} C_DIS
LIN {X -26.2456,Y -46.5905,Z 66,A -124.5499,B 24.8824,C -2.5028,E1 24.9236,E2 -151.7028} C_DIS
LIN {X -23.6222,Y -47.9737,Z 66,A -121.3683,B 24.8828,C -2.499,E1 24.9315,E2 -154.8837} C_DIS
LIN {X -21.0181,Y -49.1702,Z 66,A -118.3014,B 24.8831,C -2.4956,E1 24.9393,E2 -157.9501} C_DIS
LIN {X -19.1147,Y -49.9409,Z 66,A -115.5609,B 24.8824,C -2.5033,E1 24.9465,E2 -160.7146} C_DIS
LIN {X -14.5277,Y -51.4626,Z 66,A -111.0938,B 24.8839,C -2.4867,E1 24.9583,E2 -165.15} C_DIS
LIN {X -11.4912,Y -52.2248,Z 66,A -107.127,B 24.883,C -2.4962,E1 24.9692,E2 -169.1447} C_DIS
LIN {X -7.1232,Y -52.9976,Z 66,A -102.3071,B 24.883,C -2.4962,E1 24.9825,E2 -173.9689} C_DIS
LIN {X -2.3362,Y -53.4222,Z 66,A -97.3797,B 24.8834,C -2.4921,E1 24.9962,E2 -178.8882} C_DIS
LIN {X 0.2758,Y -53.4677,Z 66,A -95.4248,B 24.8849,C -2.4767,E1 25.0016,E2 -180.8068} C_DIS
Enddeposition()
LIN {X 0.2758,Y -53.4677,Z 66,A -95.4248,B 24.8849,C -2.4767,E1 25.0016,E2 -180.8068} C_DIS
Startdeposition()
$VEL.CP = VEL_PRINT
LIN {X -0.5849,Y -52.5122,Z 66,A -97.3689,B 24.8851,C -2.4747,E1 24.9961,E2 -178.8577} C_DIS
LIN {X -3.8859,Y -52.371,Z 66,A -100.549,B 24.8844,C -2.4821,E1 24.9873,E2 -175.6944} C_DIS
LIN {X -6.1231,Y -52.1567,Z 66,A -103.8199,B 24.8857,C -2.4678,E1 24.9781,E2 -172.3875} C_DIS
LIN {X -9.6151,Y -51.6274,Z 66,A -107.2743,B 24.8849,C -2.476,E1 24.9687,E2 -168.9492} C_DIS
LIN {X -12.6943,Y -50.9574,Z 66,A -110.3836,B 24.8842,C -2.4834,E1 24.9602,E2 -165.8535} C_DIS
LIN {X -14.6972,Y -50.4161,Z 66,A -112.7005,B 24.8842,C -2.4839,E1 24.954,E2 -163.5341} C_DIS
LIN {X -17.1253,Y -49.6439,Z 66,A -115.9538,B 24.8847,C -2.478,E1 24.9453,E2 -160.2606} C_DIS
LIN {X -19.9426,Y -48.5812,Z 66,A -118.9344,B 24.884,C -2.4862,E1 24.9376,E2 -157.2932} C_DIS
LIN {X -22.4478,Y -47.4755,Z 66,A -122.1762,B 24.884,C -2.4853,E1 24.9294,E2 -154.0411} C_DIS
LIN {X -25.8452,Y -45.7154,Z 66,A -126.0071,B 24.883,C -2.4963,E1 24.92,E2 -150.2259} C_DIS
LIN {X -27.4844,Y -44.7489,Z 66,A -128.5314,B 24.8834,C -2.492,E1 24.9139,E2 -147.6834} C_DIS
LIN {X -29.7195,Y -43.2971,Z 66,A -130.7903,B 24.882,C -2.5071,E1 24.9087,E2 -145.4531} C_DIS
LIN {X -32.4843,Y -41.2626,Z 66,A -134.8555,B 24.882,C -2.5083,E1 24.8996,E2 -141.3762} C_DIS
LIN {X -34.5785,Y -39.524,Z 66,A -137.9776,B 24.8816,C -2.5114,E1 24.893,E2 -138.2494} C_DIS
LIN {X -37.2098,Y -37.0573,Z 66,A -141.9208,B 24.8809,C -2.5193,E1 24.8851,E2 -134.3086} C_DIS
LIN {X -38.9448,Y -35.2302,Z 66,A -144.8129,B 24.8805,C -2.523,E1 24.8796,E2 -131.4125} C_DIS
LIN {X -41.1638,Y -32.6093,Z 66,A -148.6312,B 24.8798,C -2.5305,E1 24.8728,E2 -127.5944} C_DIS
LIN {X -43.2845,Y -29.7381,Z 66,A -152.3792,B 24.8787,C -2.5422,E1 24.8668,E2 -123.8561} C_DIS
LIN {X -44.9288,Y -27.1888,Z 66,A -155.5738,B 24.8777,C -2.5524,E1 24.862,E2 -120.6696} C_DIS
LIN {X -46.2356,Y -24.902,Z 66,A -158.3748,B 24.8769,C -2.5611,E1 24.8582,E2 -117.8747} C_DIS
LIN {X -47.509,Y -22.3769,Z 66,A -161.8846,B 24.8767,C -2.5632,E1 24.8539,E2 -114.3508} C_DIS
LIN {X -48.8873,Y -19.1785,Z 66,A -166.0341,B 24.8761,C -2.5688,E1 24.8496,E2 -110.1916} C_DIS
LIN {X -50.1459,Y -15.5951,Z 66,A -170.1595,B 24.8749,C -2.5811,E1 24.846,E2 -106.0722} C_DIS
LIN {X -51.3324,Y -11.0817,Z 66,A -175.2439,B 24.8734,C -2.5966,E1 24.8427,E2 -100.9949} C_DIS
LIN {X -51.9929,Y -7.3864,Z 66,A -178.8728,B 24.8715,C -2.6159,E1 24.8411,E2 -97.3907} C_DIS
LIN {X -52.3127,Y -4.6043,Z 66,A 178.0951,B 24.8705,C -2.6258,E1 24.8402,E2 -94.3639} C_DIS
LIN {X -52.5026,Y -1.1507,Z 66,A 173.9234,B 24.8699,C -2.6318,E1 24.8398,E2 -90.1816} C_DIS
LIN {X -52.4656,Y 2.2749,Z 66,A 170.5975,B 24.8682,C -2.6496,E1 24.84,E2 -86.878} C_DIS
LIN {X -52.2868,Y 4.8899,Z 66,A 167.5909,B 24.8675,C -2.6564,E1 24.8407,E2 -83.8698} C_DIS
LIN {X -51.9352,Y 7.7808,Z 66,A 164.6883,B 24.8661,C -2.6704,E1 24.8417,E2 -80.9834} C_DIS
LIN {X -51.5049,Y 10.2487,Z 66,A 161.3547,B 24.8661,C -2.6702,E1 24.8435,E2 -77.6296} C_DIS
LIN {X -50.9544,Y 12.707,Z 66,A 158.8674,B 24.8649,C -2.6825,E1 24.8451,E2 -75.1572} C_DIS
LIN {X -49.9332,Y 16.2631,Z 66,A 154.5806,B 24.864,C -2.6913,E1 24.8486,E2 -70.8666} C_DIS
LIN {X -48.877,Y 19.2056,Z 66,A 150.7005,B 24.8636,C -2.6948,E1 24.8525,E2 -66.9729} C_DIS
LIN {X -46.8138,Y 23.7968,Z 66,A 146.0986,B 24.8607,C -2.7239,E1 24.8579,E2 -62.4157} C_DIS
LIN {X -45.8856,Y 25.5404,Z 66,A 143.5584,B 24.8607,C -2.7243,E1 24.8613,E2 -59.8631} C_DIS
LIN {X -44.2176,Y 28.3306,Z 66,A 140.1381,B 24.8594,C -2.7361,E1 24.8663,E2 -56.4534} C_DIS
LIN {X -42.6763,Y 30.6024,Z 66,A 137.331,B 24.8583,C -2.747,E1 24.8707,E2 -53.6585} C_DIS
LIN {X -41.3824,Y 32.3326,Z 66,A 134.8898,B 24.8578,C -2.7518,E1 24.8749,E2 -51.2173} C_DIS
LIN {X -39.3874,Y 34.7345,Z 66,A 131.1128,B 24.8575,C -2.7548,E1 24.8817,E2 -47.4302} C_DIS
LIN {X -37.5098,Y 36.7541,Z 66,A 127.9743,B 24.8569,C -2.7601,E1 24.8878,E2 -44.2908} C_DIS
LIN {X -34.5162,Y 39.5784,Z 66,A 124.1201,B 24.8548,C -2.7801,E1 24.8957,E2 -40.4687} C_DIS
LIN {X -32.8964,Y 40.9352,Z 66,A 120.3254,B 24.8567,C -2.7621,E1 24.904,E2 -36.6168} C_DIS
LIN {X -30.0968,Y 43.0351,Z 66,A 117.1784,B 24.8548,C -2.78,E1 24.9111,E2 -33.5016} C_DIS
LIN {X -26.707,Y 45.2167,Z 66,A 113.3007,B 24.8531,C -2.7962,E1 24.9203,E2 -29.6504} C_DIS
Enddeposition()
END
